LIN {X -0.030,Y -605.100,Z 1297.595,A 0.000,B 0.000,C 90.000,E1 143.050} C_DIS
LIN {X -0.184,Y -608.244,Z 1297.593,A 0.000,B 0.000,C 90.000,E1 142.683} C_DIS
LIN {X 0.115,Y -612.176,Z 1297.590,A 0.000,B 0.000,C 90.000,E1 142.145} C_DIS
LIN {X -0.312,Y -616.700,Z 1297.586,A 0.000,B 0.000,C 90.000,E1 141.537} C_DIS
LIN {X -0.216,Y -620.888,Z 1297.583,A 0.000,B 0.000,C 90.000,E1 140.884} C_DIS
LIN {X 0.278,Y -625.462,Z 1297.578,A 0.000,B 0.000,C 90.000,E1 140.070} C_DIS
LIN {X -0.003,Y -628.392,Z 1297.576,A 0.000,B 0.000,C 90.000,E1 139.585} C_DIS
LIN {X 0.188,Y -631.713,Z 1297.572,A 0.000,B 0.000,C 90.000,E1 138.933} C_DIS
LIN {X 0.321,Y -635.448,Z 1297.568,A 0.000,B 0.000,C 90.000,E1 138.162} C_DIS
LIN {X -0.415,Y -638.910,Z 1297.564,A 0.000,B 0.000,C 90.000,E1 137.472} C_DIS
LIN {X -0.130,Y -641.202,Z 1297.561,A 0.000,B 0.000,C 90.000,E1 136.944} C_DIS
LIN {X 0.323,Y -647.787,Z 1297.552,A 0.000,B 0.000,C 90.000,E1 135.405} C_DIS
LIN {X 0.041,Y -653.046,Z 1297.546,A 0.000,B 0.000,C 90.000,E1 134.190} C_DIS
LIN {X 0.316,Y -658.199,Z 1297.539,A 0.000,B 0.000,C 90.000,E1 132.933} C_DIS
LIN {X -0.258,Y -663.302,Z 1297.532,A 0.000,B 0.000,C 90.000,E1 131.757} C_DIS
LIN {X 0.194,Y -666.234,Z 1297.528,A 0.000,B 0.000,C 90.000,E1 130.987} C_DIS
LIN {X 0.237,Y -669.954,Z 1297.522,A 0.000,B 0.000,C 90.000,E1 130.011} C_DIS
LIN {X -0.092,Y -674.260,Z 1297.516,A 0.000,B 0.000,C 90.000,E1 128.830} C_DIS
LIN {X 0.179,Y -678.263,Z 1297.509,A 0.000,B 0.000,C 90.000,E1 127.604} C_DIS
LIN {X -0.045,Y -681.139,Z 1297.504,A 0.000,B 0.000,C 90.000,E1 126.664} C_DIS
LIN {X -0.238,Y -683.829,Z 1297.498,A 0.000,B 0.000,C 90.000,E1 125.724} C_DIS
LIN {X 0.153,Y -686.315,Z 1297.493,A 0.000,B 0.000,C 90.000,E1 124.739} C_DIS
LIN {X -0.013,Y -688.024,Z 1297.489,A 0.000,B 0.000,C 90.000,E1 124.040} C_DIS
LIN {X 0.045,Y -690.041,Z 1297.484,A 0.000,B 0.000,C 90.000,E1 123.086} C_DIS
LIN {X -0.092,Y -691.353,Z 1297.480,A 0.000,B 0.000,C 90.000,E1 122.388} C_DIS
LIN {X -0.359,Y -692.948,Z 1297.475,A 0.000,B 0.000,C 90.000,E1 121.465} C_DIS
LIN {X 0.244,Y -695.108,Z 1297.467,A 0.000,B 0.000,C 90.000,E1 120.001} C_DIS
LIN {X -0.217,Y -696.091,Z 1297.463,A 0.000,B 0.000,C 90.000,E1 119.333} C_DIS
LIN {X 0.194,Y -697.188,Z 1297.458,A 0.000,B 0.000,C 90.000,E1 118.359} C_DIS
LIN {X 0.359,Y -697.753,Z 1297.454,A 0.000,B 0.000,C 90.000,E1 117.641} C_DIS
LIN {X 0.210,Y -698.075,Z 1297.450,A 0.000,B 0.000,C 90.000,E1 116.950} C_DIS
LIN {X 0.018,Y -698.206,Z 1297.445,A 0.000,B 0.000,C 90.000,E1 116.027} C_DIS
LIN {X -0.122,Y -697.858,Z 1297.441,A 0.000,B 0.000,C 90.000,E1 115.335} C_DIS
LIN {X 0.107,Y -697.472,Z 1297.438,A 0.000,B 0.000,C 90.000,E1 114.847} C_DIS
LIN {X -0.004,Y -696.661,Z 1297.436,A 0.000,B 0.000,C 90.000,E1 114.387} C_DIS
LIN {X -0.032,Y -696.081,Z 1297.434,A 0.000,B 0.000,C 90.000,E1 114.155} C_DIS
LIN {X -0.157,Y -694.510,Z 1297.432,A 0.000,B 0.000,C 90.000,E1 113.695} C_DIS
LIN {X -0.033,Y -693.891,Z 1297.431,A 0.000,B 0.000,C 90.000,E1 113.567} C_DIS
LIN {X 0.179,Y -690.653,Z 1297.428,A 0.000,B 0.000,C 90.000,E1 113.078} C_DIS
LIN {X 0.298,Y -689.612,Z 1297.428,A 0.000,B 0.000,C 90.000,E1 112.950} C_DIS
LIN {X 0.145,Y -688.043,Z 1297.427,A 0.000,B 0.000,C 90.000,E1 112.845} C_DIS
LIN {X 0.031,Y -682.035,Z 1297.425,A 0.000,B 0.000,C 90.000,E1 112.461} C_DIS
LIN {X -0.099,Y -679.841,Z 1297.424,A 0.000,B 0.000,C 90.000,E1 112.386} C_DIS
LIN {X -0.135,Y -675.300,Z 1297.424,A 0.000,B 0.000,C 90.000,E1 112.259} C_DIS
LIN {X 0.009,Y -671.699,Z 1297.423,A 0.000,B 0.000,C 90.000,E1 112.153} C_DIS
LIN {X -0.191,Y -663.966,Z 1297.423,A 0.000,B 0.000,C 90.000,E1 112.078} C_DIS
LIN {X 0.309,Y -662.814,Z 1297.423,A 0.000,B 0.000,C 90.000,E1 112.025} C_DIS
LIN {X 0.251,Y -658.276,Z 1297.422,A 0.000,B 0.000,C 90.000,E1 112.025} C_DIS
LIN {X 0.138,Y -656.155,Z 1297.422,A 0.000,B 0.000,C 90.000,E1 112.025} C_DIS
LIN {X 0.082,Y -651.599,Z 1297.422,A 0.000,B 0.000,C 90.000,E1 112.025} C_DIS
LIN {X -0.029,Y -647.834,Z 1297.422,A 0.000,B 0.000,C 90.000,E1 112.025} C_DIS
LIN {X 0.046,Y -643.398,Z 1297.422,A 0.000,B 0.000,C 90.000,E1 111.972} C_DIS
LIN {X -0.186,Y -640.160,Z 1297.422,A 0.000,B 0.000,C 90.000,E1 111.897} C_DIS
LIN {X -0.223,Y -640.102,Z 1297.422,A 0.000,B 0.000,C 90.000,E1 111.897} C_DIS
LIN {X -0.025,Y -641.829,Z 1297.420,A 0.000,B 0.000,C 90.000,E1 111.535} C_DIS
LIN {X -0.231,Y -645.606,Z 1297.417,A 0.000,B 0.000,C 90.000,E1 111.046} C_DIS
LIN {X -0.292,Y -650.402,Z 1297.413,A 0.000,B 0.000,C 90.000,E1 110.429} C_DIS
LIN {X 0.343,Y -655.261,Z 1297.409,A 0.000,B 0.000,C 90.000,E1 109.631} C_DIS
LIN {X 0.142,Y -658.719,Z 1297.406,A 0.000,B 0.000,C 90.000,E1 109.033} C_DIS
LIN {X 0.079,Y -660.661,Z 1297.404,A 0.000,B 0.000,C 90.000,E1 108.671} C_DIS
LIN {X -0.024,Y -664.077,Z 1297.400,A 0.000,B 0.000,C 90.000,E1 107.946} C_DIS
LIN {X -0.098,Y -667.037,Z 1297.396,A 0.000,B 0.000,C 90.000,E1 107.221} C_DIS
LIN {X -0.069,Y -668.785,Z 1297.393,A 0.000,B 0.000,C 90.000,E1 106.732} C_DIS
LIN {X -0.294,Y -671.049,Z 1297.389,A 0.000,B 0.000,C 90.000,E1 106.024} C_DIS
LIN {X 0.336,Y -672.875,Z 1297.385,A 0.000,B 0.000,C 90.000,E1 105.245} C_DIS
LIN {X 0.215,Y -673.985,Z 1297.382,A 0.000,B 0.000,C 90.000,E1 104.773} C_DIS
LIN {X 0.048,Y -675.282,Z 1297.378,A 0.000,B 0.000,C 90.000,E1 104.064} C_DIS
LIN {X -0.057,Y -676.027,Z 1297.375,A 0.000,B 0.000,C 90.000,E1 103.592} C_DIS
LIN {X -0.206,Y -676.735,Z 1297.372,A 0.000,B 0.000,C 90.000,E1 102.883} C_DIS
LIN {X 0.308,Y -677.148,Z 1297.368,A 0.000,B 0.000,C 90.000,E1 102.119} C_DIS
LIN {X 0.026,Y -677.120,Z 1297.364,A 0.000,B 0.000,C 90.000,E1 101.422} C_DIS
LIN {X -0.072,Y -676.885,Z 1297.361,A 0.000,B 0.000,C 90.000,E1 100.950} C_DIS
LIN {X 0.313,Y -676.130,Z 1297.357,A 0.000,B 0.000,C 90.000,E1 100.197} C_DIS
LIN {X 0.202,Y -675.321,Z 1297.354,A 0.000,B 0.000,C 90.000,E1 99.726} C_DIS
LIN {X -0.029,Y -674.316,Z 1297.352,A 0.000,B 0.000,C 90.000,E1 99.265} C_DIS
LIN {X -0.263,Y -672.938,Z 1297.349,A 0.000,B 0.000,C 90.000,E1 98.803} C_DIS
LIN {X 0.260,Y -671.215,Z 1297.346,A 0.000,B 0.000,C 90.000,E1 98.276} C_DIS
LIN {X 0.008,Y -669.140,Z 1297.344,A 0.000,B 0.000,C 90.000,E1 97.814} C_DIS
LIN {X 0.230,Y -665.625,Z 1297.339,A 0.000,B 0.000,C 90.000,E1 97.068} C_DIS
LIN {X -0.071,Y -662.116,Z 1297.336,A 0.000,B 0.000,C 90.000,E1 96.486} C_DIS
LIN {X 0.276,Y -659.164,Z 1297.333,A 0.000,B 0.000,C 90.000,E1 95.967} C_DIS
LIN {X -0.085,Y -655.897,Z 1297.331,A 0.000,B 0.000,C 90.000,E1 95.511} C_DIS
LIN {X 0.147,Y -651.287,Z 1297.327,A 0.000,B 0.000,C 90.000,E1 94.878} C_DIS
LIN {X -0.215,Y -647.287,Z 1297.324,A 0.000,B 0.000,C 90.000,E1 94.416} C_DIS
LIN {X 0.310,Y -639.394,Z 1297.320,A 0.000,B 0.000,C 90.000,E1 93.498} C_DIS
LIN {X 0.036,Y -629.758,Z 1297.314,A 0.000,B 0.000,C 90.000,E1 92.522} C_DIS
LIN {X -0.068,Y -626.245,Z 1297.312,A 0.000,B 0.000,C 90.000,E1 92.178} C_DIS
LIN {X 0.266,Y -621.098,Z 1297.309,A 0.000,B 0.000,C 90.000,E1 91.661} C_DIS
LIN {X 0.159,Y -615.486,Z 1297.307,A 0.000,B 0.000,C 90.000,E1 91.203} C_DIS
LIN {X 0.033,Y -608.005,Z 1297.304,A 0.000,B 0.000,C 90.000,E1 90.688} C_DIS
LIN {X 0.125,Y -601.709,Z 1297.302,A 0.000,B 0.000,C 90.000,E1 90.286} C_DIS
LIN {X -0.026,Y -595.069,Z 1297.300,A 0.000,B 0.000,C 90.000,E1 89.943} C_DIS
LIN {X 0.231,Y -588.114,Z 1297.298,A 0.000,B 0.000,C 90.000,E1 89.599} C_DIS
LIN {X -0.248,Y -578.956,Z 1297.296,A 0.000,B 0.000,C 90.000,E1 89.312} C_DIS
LIN {X 0.252,Y -575.828,Z 1297.295,A 0.000,B 0.000,C 90.000,E1 89.141} C_DIS
LIN {X 0.201,Y -571.918,Z 1297.294,A 0.000,B 0.000,C 90.000,E1 88.969} C_DIS
LIN {X 0.184,Y -570.507,Z 1297.294,A 0.000,B 0.000,C 90.000,E1 88.854} C_DIS
LIN {X 0.147,Y -570.464,Z 1297.294,A 0.000,B 0.000,C 90.000,E1 88.854} C_DIS
LIN {X -0.051,Y -569.912,Z 1297.293,A 0.000,B 0.000,C 90.000,E1 88.740} C_DIS
LIN {X -0.187,Y -569.791,Z 1297.291,A 0.000,B 0.000,C 90.000,E1 88.339} C_DIS
LIN {X 0.170,Y -572.199,Z 1297.274,A 0.000,B 0.000,C 90.000,E1 85.298} C_DIS
LIN {X 0.146,Y -574.318,Z 1297.263,A 0.000,B 0.000,C 90.000,E1 83.394} C_DIS
LIN {X 0.180,Y -576.536,Z 1297.253,A 0.000,B 0.000,C 90.000,E1 81.489} C_DIS
LIN {X 0.225,Y -578.520,Z 1297.244,A 0.000,B 0.000,C 90.000,E1 79.859} C_DIS
LIN {X -0.137,Y -579.666,Z 1297.238,A 0.000,B 0.000,C 90.000,E1 78.814} C_DIS
LIN {X -0.146,Y -580.931,Z 1297.230,A 0.000,B 0.000,C 90.000,E1 77.465} C_DIS
LIN {X -0.136,Y -582.120,Z 1297.223,A 0.000,B 0.000,C 90.000,E1 76.117} C_DIS
LIN {X -0.305,Y -583.309,Z 1297.214,A 0.000,B 0.000,C 90.000,E1 74.519} C_DIS
LIN {X 0.039,Y -584.186,Z 1297.206,A 0.000,B 0.000,C 90.000,E1 73.142} C_DIS
LIN {X 0.066,Y -585.263,Z 1297.198,A 0.000,B 0.000,C 90.000,E1 71.529} C_DIS
LIN {X -0.145,Y -585.939,Z 1297.192,A 0.000,B 0.000,C 90.000,E1 70.477} C_DIS
LIN {X 0.093,Y -586.922,Z 1297.183,A 0.000,B 0.000,C 90.000,E1 68.847} C_DIS
LIN {X -0.246,Y -588.232,Z 1297.171,A 0.000,B 0.000,C 90.000,E1 66.741} C_DIS
LIN {X 0.150,Y -589.357,Z 1297.162,A 0.000,B 0.000,C 90.000,E1 65.101} C_DIS
LIN {X 0.041,Y -590.511,Z 1297.153,A 0.000,B 0.000,C 90.000,E1 63.512} C_DIS
LIN {X 0.120,Y -592.082,Z 1297.143,A 0.000,B 0.000,C 90.000,E1 61.641} C_DIS
LIN {X -0.095,Y -593.382,Z 1297.135,A 0.000,B 0.000,C 90.000,E1 60.333} C_DIS
LIN {X 0.009,Y -594.730,Z 1297.128,A 0.000,B 0.000,C 90.000,E1 58.997} C_DIS
LIN {X 0.035,Y -596.340,Z 1297.119,A 0.000,B 0.000,C 90.000,E1 57.406} C_DIS
LIN {X 0.107,Y -597.490,Z 1297.113,A 0.000,B 0.000,C 90.000,E1 56.342} C_DIS
LIN {X 0.109,Y -598.850,Z 1297.106,A 0.000,B 0.000,C 90.000,E1 55.022} C_DIS
LIN {X -0.111,Y -600.333,Z 1297.097,A 0.000,B 0.000,C 90.000,E1 53.463} C_DIS
LIN {X -0.311,Y -601.668,Z 1297.088,A 0.000,B 0.000,C 90.000,E1 51.904} C_DIS
LIN {X 0.217,Y -602.537,Z 1297.082,A 0.000,B 0.000,C 90.000,E1 50.803} C_DIS
LIN {X -0.057,Y -603.473,Z 1297.074,A 0.000,B 0.000,C 90.000,E1 49.256} C_DIS
LIN {X -0.016,Y -603.749,Z 1297.071,A 0.000,B 0.000,C 90.000,E1 48.728} C_DIS
LIN {X 0.226,Y -603.990,Z 1297.066,A 0.000,B 0.000,C 90.000,E1 47.919} C_DIS
LIN {X -0.084,Y -604.366,Z 1297.058,A 0.000,B 0.000,C 90.000,E1 46.377} C_DIS
LIN {X -0.017,Y -604.520,Z 1297.052,A 0.000,B 0.000,C 90.000,E1 45.324} C_DIS
LIN {X 0.055,Y -604.463,Z 1297.046,A 0.000,B 0.000,C 90.000,E1 44.271} C_DIS
LIN {X -0.080,Y -604.111,Z 1297.039,A 0.000,B 0.000,C 90.000,E1 42.975} C_DIS
LIN {X 0.008,Y -603.839,Z 1297.033,A 0.000,B 0.000,C 90.000,E1 41.919} C_DIS
LIN {X -0.149,Y -603.531,Z 1297.029,A 0.000,B 0.000,C 90.000,E1 41.148} C_DIS
LIN {X 0.233,Y -602.687,Z 1297.018,A 0.000,B 0.000,C 90.000,E1 39.277} C_DIS
LIN {X -0.071,Y -602.062,Z 1297.013,A 0.000,B 0.000,C 90.000,E1 38.257} C_DIS
LIN {X -0.134,Y -600.871,Z 1297.005,A 0.000,B 0.000,C 90.000,E1 36.950} C_DIS
LIN {X 0.016,Y -599.578,Z 1296.999,A 0.000,B 0.000,C 90.000,E1 35.884} C_DIS
LIN {X 0.145,Y -598.081,Z 1296.994,A 0.000,B 0.000,C 90.000,E1 34.818} C_DIS
LIN {X 0.135,Y -595.738,Z 1296.986,A 0.000,B 0.000,C 90.000,E1 33.499} C_DIS
LIN {X -0.349,Y -594.062,Z 1296.982,A 0.000,B 0.000,C 90.000,E1 32.752} C_DIS
LIN {X -0.240,Y -592.810,Z 1296.979,A 0.000,B 0.000,C 90.000,E1 32.212} C_DIS
LIN {X 0.061,Y -590.612,Z 1296.974,A 0.000,B 0.000,C 90.000,E1 31.386} C_DIS
LIN {X 0.029,Y -588.195,Z 1296.970,A 0.000,B 0.000,C 90.000,E1 30.590} C_DIS
LIN {X -0.028,Y -585.262,Z 1296.966,A 0.000,B 0.000,C 90.000,E1 29.795} C_DIS
LIN {X -0.272,Y -583.140,Z 1296.963,A 0.000,B 0.000,C 90.000,E1 29.283} C_DIS
LIN {X 0.131,Y -579.545,Z 1296.958,A 0.000,B 0.000,C 90.000,E1 28.437} C_DIS
LIN {X 0.197,Y -577.635,Z 1296.956,A 0.000,B 0.000,C 90.000,E1 28.025} C_DIS
LIN {X -0.171,Y -574.033,Z 1296.952,A 0.000,B 0.000,C 90.000,E1 27.385} C_DIS
LIN {X 0.117,Y -569.415,Z 1296.948,A 0.000,B 0.000,C 90.000,E1 26.539} C_DIS
LIN {X 0.100,Y -564.275,Z 1296.943,A 0.000,B 0.000,C 90.000,E1 25.720} C_DIS
LIN {X 0.228,Y -560.522,Z 1296.940,A 0.000,B 0.000,C 90.000,E1 25.155} C_DIS
LIN {X -0.165,Y -556.580,Z 1296.937,A 0.000,B 0.000,C 90.000,E1 24.643} C_DIS
LIN {X -0.089,Y -552.362,Z 1296.934,A 0.000,B 0.000,C 90.000,E1 24.079} C_DIS
LIN {X 0.074,Y -549.001,Z 1296.931,A 0.000,B 0.000,C 90.000,E1 23.643} C_DIS
LIN {X 0.095,Y -544.241,Z 1296.928,A 0.000,B 0.000,C 90.000,E1 23.078} C_DIS
LIN {X -0.107,Y -537.173,Z 1296.924,A 0.000,B 0.000,C 90.000,E1 22.280} C_DIS
LIN {X 0.213,Y -530.692,Z 1296.920,A 0.000,B 0.000,C 90.000,E1 21.535} C_DIS
LIN {X -0.227,Y -521.569,Z 1296.914,A 0.000,B 0.000,C 90.000,E1 20.610} C_DIS
LIN {X 0.161,Y -512.498,Z 1296.909,A 0.000,B 0.000,C 90.000,E1 19.631} C_DIS
LIN {X 0.116,Y -504.674,Z 1296.905,A 0.000,B 0.000,C 90.000,E1 18.852} C_DIS
LIN {X -0.143,Y -495.008,Z 1296.900,A 0.000,B 0.000,C 90.000,E1 17.928} C_DIS
LIN {X -0.016,Y -483.925,Z 1296.894,A 0.000,B 0.000,C 90.000,E1 16.858} C_DIS
LIN {X -0.090,Y -473.781,Z 1296.889,A 0.000,B 0.000,C 90.000,E1 15.953} C_DIS
LIN {X 0.015,Y -463.432,Z 1296.883,A 0.000,B 0.000,C 90.000,E1 15.009} C_DIS
LIN {X -0.079,Y -447.415,Z 1296.875,A 0.000,B 0.000,C 90.000,E1 13.536} C_DIS
LIN {X -0.029,Y -427.454,Z 1296.864,A 0.000,B 0.000,C 90.000,E1 11.535} C_DIS
LIN {X -0.194,Y -408.819,Z 1296.853,A 0.000,B 0.000,C 90.000,E1 9.557} C_DIS
LIN {X 0.118,Y -400.386,Z 1296.848,A 0.000,B 0.000,C 90.000,E1 8.568} C_DIS
LIN {X -0.145,Y -396.849,Z 1296.845,A 0.000,B 0.000,C 90.000,E1 8.163} C_DIS
LIN {X 0.146,Y -395.306,Z 1296.844,A 0.000,B 0.000,C 90.000,E1 7.814} C_DIS
LIN {X 0.108,Y -395.286,Z 1296.844,A 0.000,B 0.000,C 90.000,E1 7.814} C_DIS
LIN {X 0.106,Y -396.353,Z 1296.843,A 0.000,B 0.000,C 90.000,E1 7.644} C_DIS
LIN {X 0.203,Y -398.732,Z 1296.841,A 0.000,B 0.000,C 90.000,E1 7.409} C_DIS
LIN {X 0.001,Y -400.479,Z 1296.841,A 0.000,B 0.000,C 90.000,E1 7.296} C_DIS
LIN {X -0.011,Y -406.290,Z 1296.839,A 0.000,B 0.000,C 90.000,E1 6.947} C_DIS
LIN {X -0.066,Y -412.341,Z 1296.837,A 0.000,B 0.000,C 90.000,E1 6.606} C_DIS
LIN {X -0.215,Y -418.697,Z 1296.834,A 0.000,B 0.000,C 90.000,E1 6.201} C_DIS
LIN {X -0.169,Y -423.565,Z 1296.832,A 0.000,B 0.000,C 90.000,E1 5.853} C_DIS
LIN {X 0.116,Y -432.755,Z 1296.828,A 0.000,B 0.000,C 90.000,E1 5.106} C_DIS
LIN {X -0.081,Y -437.351,Z 1296.826,A 0.000,B 0.000,C 90.000,E1 4.759} C_DIS
LIN {X 0.069,Y -446.607,Z 1296.822,A 0.000,B 0.000,C 90.000,E1 3.955} C_DIS
LIN {X -0.154,Y -453.959,Z 1296.818,A 0.000,B 0.000,C 90.000,E1 3.326} C_DIS
LIN {X -0.200,Y -461.137,Z 1296.815,A 0.000,B 0.000,C 90.000,E1 2.636} C_DIS
LIN {X -0.203,Y -466.756,Z 1296.811,A 0.000,B 0.000,C 90.000,E1 2.064} C_DIS
LIN {X -0.154,Y -473.457,Z 1296.807,A 0.000,B 0.000,C 90.000,E1 1.318} C_DIS
LIN {X -0.036,Y -478.418,Z 1296.804,A 0.000,B 0.000,C 90.000,E1 0.688} C_DIS
LIN {X -0.098,Y -482.096,Z 1296.801,A 0.000,B 0.000,C 90.000,E1 0.229} C_DIS
LIN {X 0.004,Y -487.458,Z 1296.797,A 0.000,B 0.000,C 90.000,E1 359.484} C_DIS
LIN {X 0.000,Y -493.503,Z 1296.792,A 0.000,B 0.000,C 90.000,E1 358.568} C_DIS
LIN {X 0.216,Y -497.387,Z 1296.789,A 0.000,B 0.000,C 90.000,E1 357.936} C_DIS
LIN {X -0.179,Y -502.545,Z 1296.784,A 0.000,B 0.000,C 90.000,E1 357.078} C_DIS
LIN {X -0.193,Y -506.613,Z 1296.780,A 0.000,B 0.000,C 90.000,E1 356.331} C_DIS
LIN {X -0.169,Y -510.442,Z 1296.775,A 0.000,B 0.000,C 90.000,E1 355.584} C_DIS
LIN {X -0.107,Y -514.022,Z 1296.771,A 0.000,B 0.000,C 90.000,E1 354.837} C_DIS
LIN {X -0.230,Y -516.705,Z 1296.768,A 0.000,B 0.000,C 90.000,E1 354.261} C_DIS
LIN {X -0.116,Y -519.816,Z 1296.764,A 0.000,B 0.000,C 90.000,E1 353.514} C_DIS
LIN {X -0.209,Y -523.311,Z 1296.759,A 0.000,B 0.000,C 90.000,E1 352.648} C_DIS
LIN {X -0.265,Y -526.526,Z 1296.754,A 0.000,B 0.000,C 90.000,E1 351.781} C_DIS
LIN {X -0.264,Y -530.268,Z 1296.748,A 0.000,B 0.000,C 90.000,E1 350.622} C_DIS
LIN {X -0.158,Y -532.820,Z 1296.743,A 0.000,B 0.000,C 90.000,E1 349.746} C_DIS
LIN {X 0.033,Y -535.871,Z 1296.737,A 0.000,B 0.000,C 90.000,E1 348.578} C_DIS
LIN {X 0.207,Y -537.895,Z 1296.732,A 0.000,B 0.000,C 90.000,E1 347.701} C_DIS
LIN {X -0.125,Y -539.628,Z 1296.727,A 0.000,B 0.000,C 90.000,E1 346.881} C_DIS
LIN {X -0.240,Y -541.622,Z 1296.721,A 0.000,B 0.000,C 90.000,E1 345.755} C_DIS
LIN {X -0.093,Y -542.514,Z 1296.718,A 0.000,B 0.000,C 90.000,E1 345.172} C_DIS
LIN {X -0.249,Y -543.546,Z 1296.713,A 0.000,B 0.000,C 90.000,E1 344.338} C_DIS
LIN {X 0.129,Y -544.404,Z 1296.708,A 0.000,B 0.000,C 90.000,E1 343.449} C_DIS
LIN {X 0.154,Y -545.096,Z 1296.703,A 0.000,B 0.000,C 90.000,E1 342.598} C_DIS
LIN {X 0.024,Y -545.466,Z 1296.699,A 0.000,B 0.000,C 90.000,E1 341.764} C_DIS
LIN {X 0.068,Y -545.510,Z 1296.694,A 0.000,B 0.000,C 90.000,E1 340.913} C_DIS
LIN {X 0.114,Y -545.290,Z 1296.689,A 0.000,B 0.000,C 90.000,E1 340.061} C_DIS
LIN {X -0.091,Y -544.955,Z 1296.686,A 0.000,B 0.000,C 90.000,E1 339.518} C_DIS
LIN {X 0.142,Y -544.243,Z 1296.682,A 0.000,B 0.000,C 90.000,E1 338.646} C_DIS
LIN {X -0.318,Y -543.959,Z 1296.680,A 0.000,B 0.000,C 90.000,E1 338.411} C_DIS
LIN {X 0.122,Y -541.386,Z 1296.671,A 0.000,B 0.000,C 90.000,E1 336.666} C_DIS
LIN {X -0.172,Y -539.466,Z 1296.666,A 0.000,B 0.000,C 90.000,E1 335.845} C_DIS
LIN {X 0.276,Y -537.998,Z 1296.663,A 0.000,B 0.000,C 90.000,E1 335.229} C_DIS
LIN {X -0.055,Y -535.645,Z 1296.658,A 0.000,B 0.000,C 90.000,E1 334.409} C_DIS
LIN {X 0.018,Y -531.934,Z 1296.651,A 0.000,B 0.000,C 90.000,E1 333.256} C_DIS
LIN {X 0.037,Y -528.228,Z 1296.645,A 0.000,B 0.000,C 90.000,E1 332.103} C_DIS
LIN {X -0.158,Y -525.084,Z 1296.640,A 0.000,B 0.000,C 90.000,E1 331.257} C_DIS
LIN {X 0.030,Y -522.114,Z 1296.636,A 0.000,B 0.000,C 90.000,E1 330.511} C_DIS
LIN {X -0.067,Y -518.892,Z 1296.632,A 0.000,B 0.000,C 90.000,E1 329.793} C_DIS
LIN {X 0.162,Y -513.915,Z 1296.626,A 0.000,B 0.000,C 90.000,E1 328.742} C_DIS
LIN {X 0.247,Y -510.206,Z 1296.622,A 0.000,B 0.000,C 90.000,E1 327.995} C_DIS
LIN {X 0.004,Y -504.500,Z 1296.616,A 0.000,B 0.000,C 90.000,E1 326.834} C_DIS
LIN {X 0.086,Y -500.941,Z 1296.611,A 0.000,B 0.000,C 90.000,E1 325.928} C_DIS
LIN {X -0.031,Y -499.901,Z 1296.609,A 0.000,B 0.000,C 90.000,E1 325.642} C_DIS
LIN {X -0.277,Y -497.630,Z 1296.604,A 0.000,B 0.000,C 90.000,E1 324.769} C_DIS
LIN {X 0.023,Y -496.098,Z 1296.599,A 0.000,B 0.000,C 90.000,E1 323.829} C_DIS
LIN {X 0.034,Y -494.696,Z 1296.591,A 0.000,B 0.000,C 90.000,E1 322.316} C_DIS
LIN {X 0.162,Y -494.242,Z 1296.584,A 0.000,B 0.000,C 90.000,E1 321.090} C_DIS
LIN {X -0.205,Y -494.321,Z 1296.569,A 0.000,B 0.000,C 90.000,E1 318.405} C_DIS
LIN {X 0.021,Y -494.491,Z 1296.560,A 0.000,B 0.000,C 90.000,E1 316.863} C_DIS
LIN {X 0.048,Y -494.625,Z 1296.554,A 0.000,B 0.000,C 90.000,E1 315.648} C_DIS
LIN {X -0.101,Y -494.374,Z 1296.549,A 0.000,B 0.000,C 90.000,E1 314.757} C_DIS
LIN {X 0.263,Y -493.971,Z 1296.545,A 0.000,B 0.000,C 90.000,E1 314.109} C_DIS
LIN {X -0.075,Y -493.312,Z 1296.542,A 0.000,B 0.000,C 90.000,E1 313.542} C_DIS
LIN {X 0.102,Y -492.831,Z 1296.540,A 0.000,B 0.000,C 90.000,E1 313.218} C_DIS
LIN {X -0.059,Y -492.218,Z 1296.539,A 0.000,B 0.000,C 90.000,E1 312.933} C_DIS
LIN {X 0.115,Y -491.395,Z 1296.537,A 0.000,B 0.000,C 90.000,E1 312.609} C_DIS
LIN {X 0.200,Y -490.846,Z 1296.536,A 0.000,B 0.000,C 90.000,E1 312.447} C_DIS
LIN {X -0.046,Y -490.118,Z 1296.535,A 0.000,B 0.000,C 90.000,E1 312.324} C_DIS
LIN {X 0.229,Y -480.831,Z 1296.528,A 0.000,B 0.000,C 90.000,E1 311.067} C_DIS
LIN {X 0.080,Y -463.374,Z 1296.515,A 0.000,B 0.000,C 90.000,E1 308.588} C_DIS
LIN {X 0.214,Y -447.591,Z 1296.500,A 0.000,B 0.000,C 90.000,E1 306.011} C_DIS
LIN {X 0.052,Y -432.542,Z 1296.485,A 0.000,B 0.000,C 90.000,E1 303.245} C_DIS
LIN {X -0.081,Y -419.160,Z 1296.469,A 0.000,B 0.000,C 90.000,E1 300.413} C_DIS
LIN {X -0.139,Y -407.347,Z 1296.453,A 0.000,B 0.000,C 90.000,E1 297.513} C_DIS
LIN {X -0.160,Y -399.156,Z 1296.440,A 0.000,B 0.000,C 90.000,E1 295.207} C_DIS
LIN {X 0.163,Y -399.138,Z 1296.440,A 0.000,B 0.000,C 90.000,E1 295.155} C_DIS
LIN {X 0.076,Y -401.525,Z 1296.427,A 0.000,B 0.000,C 90.000,E1 292.770} C_DIS
LIN {X 0.109,Y -401.877,Z 1296.421,A 0.000,B 0.000,C 90.000,E1 291.716} C_DIS
LIN {X -0.168,Y -404.596,Z 1296.396,A 0.000,B 0.000,C 90.000,E1 287.221} C_DIS
LIN {X -0.068,Y -404.758,Z 1296.394,A 0.000,B 0.000,C 90.000,E1 286.858} C_DIS
LIN {X -0.161,Y -406.059,Z 1296.365,A 0.000,B 0.000,C 90.000,E1 281.658} C_DIS
LIN {X -0.071,Y -406.123,Z 1296.363,A 0.000,B 0.000,C 90.000,E1 281.299} C_DIS
LIN {X -0.041,Y -405.663,Z 1296.334,A 0.000,B 0.000,C 90.000,E1 276.087} C_DIS
LIN {X -0.036,Y -405.577,Z 1296.332,A 0.000,B 0.000,C 90.000,E1 275.739} C_DIS
LIN {X 0.038,Y -403.537,Z 1296.305,A 0.000,B 0.000,C 90.000,E1 270.859} C_DIS
LIN {X -0.027,Y -403.004,Z 1296.301,A 0.000,B 0.000,C 90.000,E1 270.172} C_DIS
LIN {X 0.193,Y -398.991,Z 1296.272,A 0.000,B 0.000,C 90.000,E1 264.894} C_DIS
LIN {X -0.043,Y -392.898,Z 1296.240,A 0.000,B 0.000,C 90.000,E1 259.285} C_DIS
LIN {X -0.096,Y -391.246,Z 1296.235,A 0.000,B 0.000,C 90.000,E1 258.229} C_DIS
LIN {X 0.098,Y -385.339,Z 1296.209,A 0.000,B 0.000,C 90.000,E1 253.559} C_DIS
LIN {X 0.120,Y -384.904,Z 1296.207,A 0.000,B 0.000,C 90.000,E1 253.196} C_DIS
LIN {X 0.120,Y -381.655,Z 1296.196,A 0.000,B 0.000,C 90.000,E1 251.329} C_DIS
LIN {X 0.082,Y -381.665,Z 1296.196,A 0.000,B 0.000,C 90.000,E1 251.329} C_DIS
LIN {X 0.178,Y -390.790,Z 1296.177,A 0.000,B 0.000,C 90.000,E1 247.794} C_DIS
LIN {X -0.208,Y -400.781,Z 1296.159,A 0.000,B 0.000,C 90.000,E1 244.665} C_DIS
LIN {X -0.081,Y -411.695,Z 1296.143,A 0.000,B 0.000,C 90.000,E1 241.691} C_DIS
LIN {X -0.078,Y -424.135,Z 1296.127,A 0.000,B 0.000,C 90.000,E1 238.791} C_DIS
LIN {X 0.086,Y -438.192,Z 1296.111,A 0.000,B 0.000,C 90.000,E1 235.928} C_DIS
LIN {X -0.078,Y -452.017,Z 1296.097,A 0.000,B 0.000,C 90.000,E1 233.497} C_DIS
LIN {X -0.087,Y -452.738,Z 1296.096,A 0.000,B 0.000,C 90.000,E1 233.336} C_DIS
LIN {X 0.267,Y -453.254,Z 1296.095,A 0.000,B 0.000,C 90.000,E1 233.130} C_DIS
LIN {X -0.016,Y -453.988,Z 1296.094,A 0.000,B 0.000,C 90.000,E1 232.844} C_DIS
LIN {X -0.298,Y -454.503,Z 1296.092,A 0.000,B 0.000,C 90.000,E1 232.557} C_DIS
LIN {X -0.217,Y -455.156,Z 1296.088,A 0.000,B 0.000,C 90.000,E1 231.904} C_DIS
LIN {X -0.120,Y -455.578,Z 1296.083,A 0.000,B 0.000,C 90.000,E1 230.928} C_DIS
LIN {X -0.011,Y -455.552,Z 1296.078,A 0.000,B 0.000,C 90.000,E1 229.952} C_DIS
LIN {X -0.086,Y -454.876,Z 1296.065,A 0.000,B 0.000,C 90.000,E1 227.715} C_DIS
LIN {X -0.270,Y -454.436,Z 1296.054,A 0.000,B 0.000,C 90.000,E1 225.810} C_DIS
LIN {X -0.121,Y -454.299,Z 1296.042,A 0.000,B 0.000,C 90.000,E1 223.542} C_DIS
LIN {X 0.023,Y -455.854,Z 1296.013,A 0.000,B 0.000,C 90.000,E1 218.382} C_DIS
LIN {X 0.037,Y -457.124,Z 1296.003,A 0.000,B 0.000,C 90.000,E1 216.457} C_DIS
LIN {X -0.224,Y -459.810,Z 1295.985,A 0.000,B 0.000,C 90.000,E1 213.293} C_DIS
LIN {X 0.027,Y -463.273,Z 1295.967,A 0.000,B 0.000,C 90.000,E1 210.079} C_DIS
LIN {X 0.086,Y -465.311,Z 1295.958,A 0.000,B 0.000,C 90.000,E1 208.487} C_DIS
LIN {X -0.089,Y -469.122,Z 1295.943,A 0.000,B 0.000,C 90.000,E1 205.668} C_DIS
LIN {X 0.060,Y -471.422,Z 1295.934,A 0.000,B 0.000,C 90.000,E1 204.079} C_DIS
LIN {X 0.021,Y -474.125,Z 1295.923,A 0.000,B 0.000,C 90.000,E1 202.206} C_DIS
LIN {X -0.143,Y -476.966,Z 1295.913,A 0.000,B 0.000,C 90.000,E1 200.355} C_DIS
LIN {X 0.049,Y -479.406,Z 1295.904,A 0.000,B 0.000,C 90.000,E1 198.779} C_DIS
LIN {X 0.145,Y -481.900,Z 1295.896,A 0.000,B 0.000,C 90.000,E1 197.221} C_DIS
LIN {X -0.176,Y -484.438,Z 1295.887,A 0.000,B 0.000,C 90.000,E1 195.717} C_DIS
LIN {X -0.125,Y -486.910,Z 1295.879,A 0.000,B 0.000,C 90.000,E1 194.175} C_DIS
LIN {X -0.142,Y -489.429,Z 1295.870,A 0.000,B 0.000,C 90.000,E1 192.647} C_DIS
LIN {X 0.167,Y -492.369,Z 1295.860,A 0.000,B 0.000,C 90.000,E1 190.782} C_DIS
LIN {X 0.157,Y -494.834,Z 1295.852,A 0.000,B 0.000,C 90.000,E1 189.265} C_DIS
LIN {X 0.107,Y -497.287,Z 1295.843,A 0.000,B 0.000,C 90.000,E1 187.757} C_DIS
LIN {X -0.053,Y -500.128,Z 1295.833,A 0.000,B 0.000,C 90.000,E1 185.967} C_DIS
LIN {X 0.004,Y -501.996,Z 1295.827,A 0.000,B 0.000,C 90.000,E1 184.759} C_DIS
LIN {X 0.242,Y -505.046,Z 1295.815,A 0.000,B 0.000,C 90.000,E1 182.636} C_DIS
LIN {X -0.169,Y -506.619,Z 1295.808,A 0.000,B 0.000,C 90.000,E1 181.489} C_DIS
LIN {X -0.159,Y -508.417,Z 1295.800,A 0.000,B 0.000,C 90.000,E1 180.000} C_DIS
LIN {X -0.024,Y -509.682,Z 1295.793,A 0.000,B 0.000,C 90.000,E1 178.797} C_DIS
LIN {X 0.142,Y -510.735,Z 1295.787,A 0.000,B 0.000,C 90.000,E1 177.593} C_DIS
LIN {X -0.184,Y -511.719,Z 1295.780,A 0.000,B 0.000,C 90.000,E1 176.445} C_DIS
LIN {X 0.097,Y -512.241,Z 1295.775,A 0.000,B 0.000,C 90.000,E1 175.527} C_DIS
LIN {X -0.171,Y -512.768,Z 1295.769,A 0.000,B 0.000,C 90.000,E1 174.375} C_DIS
LIN {X 0.077,Y -512.987,Z 1295.762,A 0.000,B 0.000,C 90.000,E1 173.166} C_DIS
LIN {X -0.119,Y -512.937,Z 1295.756,A 0.000,B 0.000,C 90.000,E1 172.008} C_DIS
LIN {X 0.223,Y -512.634,Z 1295.751,A 0.000,B 0.000,C 90.000,E1 171.084} C_DIS
LIN {X 0.017,Y -511.872,Z 1295.744,A 0.000,B 0.000,C 90.000,E1 169.926} C_DIS
LIN {X -0.111,Y -510.857,Z 1295.738,A 0.000,B 0.000,C 90.000,E1 168.757} C_DIS
LIN {X -0.216,Y -509.724,Z 1295.733,A 0.000,B 0.000,C 90.000,E1 167.881} C_DIS
LIN {X -0.182,Y -508.876,Z 1295.729,A 0.000,B 0.000,C 90.000,E1 167.285} C_DIS
LIN {X 0.136,Y -506.863,Z 1295.723,A 0.000,B 0.000,C 90.000,E1 166.061} C_DIS
LIN {X 0.156,Y -505.632,Z 1295.719,A 0.000,B 0.000,C 90.000,E1 165.463} C_DIS
LIN {X 0.045,Y -503.186,Z 1295.713,A 0.000,B 0.000,C 90.000,E1 164.283} C_DIS
LIN {X 0.031,Y -500.598,Z 1295.706,A 0.000,B 0.000,C 90.000,E1 163.087} C_DIS
LIN {X 0.132,Y -497.598,Z 1295.699,A 0.000,B 0.000,C 90.000,E1 161.873} C_DIS
LIN {X 0.080,Y -493.755,Z 1295.691,A 0.000,B 0.000,C 90.000,E1 160.369} C_DIS
LIN {X 0.110,Y -489.657,Z 1295.683,A 0.000,B 0.000,C 90.000,E1 158.847} C_DIS
LIN {X -0.256,Y -487.784,Z 1295.677,A 0.000,B 0.000,C 90.000,E1 157.975} C_DIS
LIN {X -0.209,Y -487.143,Z 1295.674,A 0.000,B 0.000,C 90.000,E1 157.358} C_DIS
LIN {X -0.188,Y -487.149,Z 1295.672,A 0.000,B 0.000,C 90.000,E1 157.050} C_DIS
LIN {X -0.170,Y -487.657,Z 1295.671,A 0.000,B 0.000,C 90.000,E1 156.741} C_DIS
LIN {X -0.146,Y -489.766,Z 1295.667,A 0.000,B 0.000,C 90.000,E1 155.973} C_DIS
LIN {X 0.031,Y -491.600,Z 1295.665,A 0.000,B 0.000,C 90.000,E1 155.613} C_DIS
LIN {X -0.178,Y -493.182,Z 1295.664,A 0.000,B 0.000,C 90.000,E1 155.485} C_DIS
LIN {X 0.061,Y -494.422,Z 1295.663,A 0.000,B 0.000,C 90.000,E1 155.305} C_DIS
LIN {X 0.064,Y -495.469,Z 1295.662,A 0.000,B 0.000,C 90.000,E1 155.153} C_DIS
LIN {X -0.141,Y -496.751,Z 1295.661,A 0.000,B 0.000,C 90.000,E1 155.025} C_DIS
LIN {X 0.005,Y -498.389,Z 1295.660,A 0.000,B 0.000,C 90.000,E1 154.845} C_DIS
LIN {X -0.185,Y -500.801,Z 1295.659,A 0.000,B 0.000,C 90.000,E1 154.588} C_DIS
LIN {X 0.118,Y -504.077,Z 1295.657,A 0.000,B 0.000,C 90.000,E1 154.229} C_DIS
LIN {X 0.192,Y -510.392,Z 1295.653,A 0.000,B 0.000,C 90.000,E1 153.512} C_DIS
LIN {X -0.061,Y -515.397,Z 1295.650,A 0.000,B 0.000,C 90.000,E1 152.948} C_DIS
LIN {X -0.051,Y -519.927,Z 1295.646,A 0.000,B 0.000,C 90.000,E1 152.359} C_DIS
LIN {X 0.159,Y -523.160,Z 1295.644,A 0.000,B 0.000,C 90.000,E1 151.897} C_DIS
LIN {X 0.233,Y -526.955,Z 1295.641,A 0.000,B 0.000,C 90.000,E1 151.307} C_DIS
LIN {X 0.184,Y -530.973,Z 1295.637,A 0.000,B 0.000,C 90.000,E1 150.589} C_DIS
LIN {X -0.147,Y -533.775,Z 1295.634,A 0.000,B 0.000,C 90.000,E1 150.049} C_DIS
LIN {X 0.023,Y -534.905,Z 1295.632,A 0.000,B 0.000,C 90.000,E1 149.744} C_DIS
LIN {X 0.003,Y -536.504,Z 1295.630,A 0.000,B 0.000,C 90.000,E1 149.459} C_DIS
LIN {X 0.178,Y -538.050,Z 1295.629,A 0.000,B 0.000,C 90.000,E1 149.203} C_DIS
LIN {X 0.036,Y -538.805,Z 1295.628,A 0.000,B 0.000,C 90.000,E1 149.076} C_DIS
LIN {X -0.106,Y -539.368,Z 1295.627,A 0.000,B 0.000,C 90.000,E1 148.948} C_DIS
LIN {X 0.033,Y -540.288,Z 1295.627,A 0.000,B 0.000,C 90.000,E1 148.791} C_DIS
LIN {X -0.106,Y -541.600,Z 1295.626,A 0.000,B 0.000,C 90.000,E1 148.663} C_DIS
LIN {X -0.251,Y -548.104,Z 1295.623,A 0.000,B 0.000,C 90.000,E1 148.201} C_DIS
LIN {X 0.124,Y -561.740,Z 1295.618,A 0.000,B 0.000,C 90.000,E1 147.248} C_DIS
LIN {X 0.164,Y -568.960,Z 1295.615,A 0.000,B 0.000,C 90.000,E1 146.707} C_DIS
LIN {X 0.048,Y -576.390,Z 1295.612,A 0.000,B 0.000,C 90.000,E1 146.167} C_DIS
LIN {X -0.005,Y -581.940,Z 1295.610,A 0.000,B 0.000,C 90.000,E1 145.722} C_DIS
LIN {X -0.089,Y -590.238,Z 1295.606,A 0.000,B 0.000,C 90.000,E1 145.022} C_DIS
LIN {X 0.123,Y -594.047,Z 1295.604,A 0.000,B 0.000,C 90.000,E1 144.642} C_DIS
LIN {X 0.277,Y -600.295,Z 1295.600,A 0.000,B 0.000,C 90.000,E1 143.989} C_DIS
LIN {X 0.006,Y -603.813,Z 1295.598,A 0.000,B 0.000,C 90.000,E1 143.623} C_DIS
LIN {X 0.213,Y -607.108,Z 1295.596,A 0.000,B 0.000,C 90.000,E1 143.210} C_DIS
LIN {X 0.229,Y -612.050,Z 1295.592,A 0.000,B 0.000,C 90.000,E1 142.557} C_DIS
LIN {X -0.009,Y -614.832,Z 1295.590,A 0.000,B 0.000,C 90.000,E1 142.190} C_DIS
LIN {X 0.110,Y -618.288,Z 1295.587,A 0.000,B 0.000,C 90.000,E1 141.662} C_DIS
LIN {X -0.326,Y -623.966,Z 1295.582,A 0.000,B 0.000,C 90.000,E1 140.803} C_DIS
LIN {X -0.170,Y -627.587,Z 1295.579,A 0.000,B 0.000,C 90.000,E1 140.150} C_DIS
LIN {X 0.040,Y -630.325,Z 1295.576,A 0.000,B 0.000,C 90.000,E1 139.622} C_DIS
LIN {X -0.349,Y -634.779,Z 1295.571,A 0.000,B 0.000,C 90.000,E1 138.771} C_DIS
LIN {X -0.191,Y -638.234,Z 1295.567,A 0.000,B 0.000,C 90.000,E1 138.000} C_DIS
LIN {X -0.083,Y -642.650,Z 1295.561,A 0.000,B 0.000,C 90.000,E1 136.986} C_DIS
LIN {X -0.047,Y -648.938,Z 1295.553,A 0.000,B 0.000,C 90.000,E1 135.486} C_DIS
LIN {X -0.312,Y -654.028,Z 1295.546,A 0.000,B 0.000,C 90.000,E1 134.271} C_DIS
LIN {X -0.025,Y -659.012,Z 1295.539,A 0.000,B 0.000,C 90.000,E1 133.014} C_DIS
LIN {X 0.350,Y -663.946,Z 1295.532,A 0.000,B 0.000,C 90.000,E1 131.757} C_DIS
LIN {X -0.120,Y -665.887,Z 1295.530,A 0.000,B 0.000,C 90.000,E1 131.310} C_DIS
LIN {X -0.081,Y -670.446,Z 1295.523,A 0.000,B 0.000,C 90.000,E1 130.092} C_DIS
LIN {X 0.022,Y -674.668,Z 1295.516,A 0.000,B 0.000,C 90.000,E1 128.874} C_DIS
LIN {X 0.290,Y -678.600,Z 1295.509,A 0.000,B 0.000,C 90.000,E1 127.649} C_DIS
LIN {X 0.065,Y -681.458,Z 1295.504,A 0.000,B 0.000,C 90.000,E1 126.710} C_DIS
LIN {X 0.024,Y -684.120,Z 1295.499,A 0.000,B 0.000,C 90.000,E1 125.758} C_DIS
LIN {X -0.135,Y -686.598,Z 1295.493,A 0.000,B 0.000,C 90.000,E1 124.818} C_DIS
LIN {X -0.296,Y -688.294,Z 1295.490,A 0.000,B 0.000,C 90.000,E1 124.119} C_DIS
LIN {X -0.232,Y -690.312,Z 1295.484,A 0.000,B 0.000,C 90.000,E1 123.166} C_DIS
LIN {X -0.140,Y -692.062,Z 1295.479,A 0.000,B 0.000,C 90.000,E1 122.212} C_DIS
LIN {X -0.029,Y -693.583,Z 1295.474,A 0.000,B 0.000,C 90.000,E1 121.258} C_DIS
LIN {X -0.365,Y -695.766,Z 1295.466,A 0.000,B 0.000,C 90.000,E1 119.873} C_DIS
LIN {X 0.045,Y -697.005,Z 1295.461,A 0.000,B 0.000,C 90.000,E1 118.899} C_DIS
LIN {X -0.401,Y -697.752,Z 1295.457,A 0.000,B 0.000,C 90.000,E1 118.231} C_DIS
LIN {X -0.231,Y -698.275,Z 1295.453,A 0.000,B 0.000,C 90.000,E1 117.513} C_DIS
LIN {X -0.059,Y -698.569,Z 1295.449,A 0.000,B 0.000,C 90.000,E1 116.796} C_DIS
LIN {X -0.198,Y -698.656,Z 1295.445,A 0.000,B 0.000,C 90.000,E1 116.104} C_DIS
LIN {X -0.332,Y -698.385,Z 1295.441,A 0.000,B 0.000,C 90.000,E1 115.412} C_DIS
LIN {X 0.199,Y -698.000,Z 1295.438,A 0.000,B 0.000,C 90.000,E1 114.899} C_DIS
LIN {X -0.200,Y -697.254,Z 1295.436,A 0.000,B 0.000,C 90.000,E1 114.463} C_DIS
LIN {X 0.061,Y -696.801,Z 1295.435,A 0.000,B 0.000,C 90.000,E1 114.207} C_DIS
LIN {X -0.343,Y -695.202,Z 1295.432,A 0.000,B 0.000,C 90.000,E1 113.770} C_DIS
LIN {X -0.089,Y -694.028,Z 1295.431,A 0.000,B 0.000,C 90.000,E1 113.515} C_DIS
LIN {X 0.127,Y -690.723,Z 1295.428,A 0.000,B 0.000,C 90.000,E1 113.025} C_DIS
LIN {X 0.246,Y -689.516,Z 1295.427,A 0.000,B 0.000,C 90.000,E1 112.898} C_DIS
LIN {X 0.002,Y -683.395,Z 1295.425,A 0.000,B 0.000,C 90.000,E1 112.514} C_DIS
LIN {X 0.131,Y -681.668,Z 1295.425,A 0.000,B 0.000,C 90.000,E1 112.408} C_DIS
LIN {X 0.011,Y -679.050,Z 1295.424,A 0.000,B 0.000,C 90.000,E1 112.333} C_DIS
LIN {X 0.061,Y -672.306,Z 1295.423,A 0.000,B 0.000,C 90.000,E1 112.153} C_DIS
LIN {X 0.140,Y -669.432,Z 1295.423,A 0.000,B 0.000,C 90.000,E1 112.099} C_DIS
LIN {X 0.241,Y -662.471,Z 1295.422,A 0.000,B 0.000,C 90.000,E1 112.025} C_DIS
LIN {X 0.182,Y -655.785,Z 1295.422,A 0.000,B 0.000,C 90.000,E1 112.025} C_DIS
LIN {X 0.126,Y -648.917,Z 1295.422,A 0.000,B 0.000,C 90.000,E1 112.025} C_DIS
LIN {X -0.148,Y -644.776,Z 1295.422,A 0.000,B 0.000,C 90.000,E1 112.025} C_DIS
LIN {X 0.021,Y -642.552,Z 1295.422,A 0.000,B 0.000,C 90.000,E1 111.972} C_DIS
LIN {X -0.072,Y -639.738,Z 1295.422,A 0.000,B 0.000,C 90.000,E1 111.897} C_DIS
LIN {X -0.109,Y -639.729,Z 1295.422,A 0.000,B 0.000,C 90.000,E1 111.897} C_DIS
LIN {X -0.171,Y -641.257,Z 1295.420,A 0.000,B 0.000,C 90.000,E1 111.589} C_DIS
LIN {X -0.181,Y -642.399,Z 1295.419,A 0.000,B 0.000,C 90.000,E1 111.408} C_DIS
LIN {X 0.185,Y -649.634,Z 1295.414,A 0.000,B 0.000,C 90.000,E1 110.429} C_DIS
LIN {X 0.076,Y -652.160,Z 1295.412,A 0.000,B 0.000,C 90.000,E1 110.066} C_DIS
LIN {X 0.024,Y -655.335,Z 1295.409,A 0.000,B 0.000,C 90.000,E1 109.577} C_DIS
LIN {X -0.079,Y -660.030,Z 1295.404,A 0.000,B 0.000,C 90.000,E1 108.725} C_DIS
LIN {X -0.190,Y -663.489,Z 1295.400,A 0.000,B 0.000,C 90.000,E1 108.000} C_DIS
LIN {X -0.273,Y -666.484,Z 1295.396,A 0.000,B 0.000,C 90.000,E1 107.275} C_DIS
LIN {X 0.197,Y -668.294,Z 1295.393,A 0.000,B 0.000,C 90.000,E1 106.749} C_DIS
LIN {X 0.162,Y -670.608,Z 1295.389,A 0.000,B 0.000,C 90.000,E1 106.024} C_DIS
LIN {X 0.140,Y -672.470,Z 1295.385,A 0.000,B 0.000,C 90.000,E1 105.300} C_DIS
LIN {X -0.046,Y -674.081,Z 1295.381,A 0.000,B 0.000,C 90.000,E1 104.592} C_DIS
LIN {X -0.160,Y -674.913,Z 1295.378,A 0.000,B 0.000,C 90.000,E1 104.120} C_DIS
LIN {X 0.337,Y -675.966,Z 1295.374,A 0.000,B 0.000,C 90.000,E1 103.355} C_DIS
LIN {X 0.186,Y -676.594,Z 1295.370,A 0.000,B 0.000,C 90.000,E1 102.647} C_DIS
LIN {X -0.104,Y -676.847,Z 1295.366,A 0.000,B 0.000,C 90.000,E1 101.951} C_DIS
LIN {X -0.201,Y -676.800,Z 1295.364,A 0.000,B 0.000,C 90.000,E1 101.478} C_DIS
LIN {X 0.362,Y -676.565,Z 1295.361,A 0.000,B 0.000,C 90.000,E1 100.950} C_DIS
LIN {X 0.079,Y -675.837,Z 1295.357,A 0.000,B 0.000,C 90.000,E1 100.254} C_DIS
LIN {X -0.150,Y -675.086,Z 1295.354,A 0.000,B 0.000,C 90.000,E1 99.792} C_DIS
LIN {X -0.269,Y -674.062,Z 1295.352,A 0.000,B 0.000,C 90.000,E1 99.321} C_DIS
LIN {X 0.161,Y -672.688,Z 1295.349,A 0.000,B 0.000,C 90.000,E1 98.803} C_DIS
LIN {X -0.081,Y -671.024,Z 1295.346,A 0.000,B 0.000,C 90.000,E1 98.341} C_DIS
LIN {X -0.236,Y -669.006,Z 1295.344,A 0.000,B 0.000,C 90.000,E1 97.871} C_DIS
LIN {X 0.162,Y -666.691,Z 1295.341,A 0.000,B 0.000,C 90.000,E1 97.352} C_DIS
LIN {X -0.024,Y -664.803,Z 1295.339,A 0.000,B 0.000,C 90.000,E1 97.004} C_DIS
LIN {X 0.247,Y -661.254,Z 1295.336,A 0.000,B 0.000,C 90.000,E1 96.372} C_DIS
LIN {X -0.067,Y -658.210,Z 1295.333,A 0.000,B 0.000,C 90.000,E1 95.910} C_DIS
LIN {X 0.251,Y -654.780,Z 1295.330,A 0.000,B 0.000,C 90.000,E1 95.391} C_DIS
LIN {X -0.268,Y -650.058,Z 1295.327,A 0.000,B 0.000,C 90.000,E1 94.821} C_DIS
LIN {X 0.108,Y -647.049,Z 1295.325,A 0.000,B 0.000,C 90.000,E1 94.416} C_DIS
LIN {X 0.108,Y -640.263,Z 1295.320,A 0.000,B 0.000,C 90.000,E1 93.669} C_DIS
LIN {X 0.106,Y -633.016,Z 1295.316,A 0.000,B 0.000,C 90.000,E1 92.922} C_DIS
LIN {X 0.134,Y -625.663,Z 1295.312,A 0.000,B 0.000,C 90.000,E1 92.178} C_DIS
LIN {X -0.153,Y -620.435,Z 1295.310,A 0.000,B 0.000,C 90.000,E1 91.718} C_DIS
LIN {X -0.271,Y -616.225,Z 1295.307,A 0.000,B 0.000,C 90.000,E1 91.375} C_DIS
LIN {X 0.277,Y -608.996,Z 1295.305,A 0.000,B 0.000,C 90.000,E1 90.802} C_DIS
LIN {X 0.218,Y -602.580,Z 1295.302,A 0.000,B 0.000,C 90.000,E1 90.401} C_DIS
LIN {X -0.024,Y -596.006,Z 1295.300,A 0.000,B 0.000,C 90.000,E1 90.057} C_DIS
LIN {X 0.109,Y -589.041,Z 1295.298,A 0.000,B 0.000,C 90.000,E1 89.714} C_DIS
LIN {X 0.088,Y -581.441,Z 1295.297,A 0.000,B 0.000,C 90.000,E1 89.427} C_DIS
LIN {X -0.036,Y -576.223,Z 1295.296,A 0.000,B 0.000,C 90.000,E1 89.255} C_DIS
LIN {X -0.239,Y -572.211,Z 1295.295,A 0.000,B 0.000,C 90.000,E1 89.083} C_DIS
LIN {X -0.243,Y -570.188,Z 1295.294,A 0.000,B 0.000,C 90.000,E1 88.912} C_DIS
LIN {X -0.282,Y -570.171,Z 1295.294,A 0.000,B 0.000,C 90.000,E1 88.912} C_DIS
LIN {X -0.179,Y -569.870,Z 1295.293,A 0.000,B 0.000,C 90.000,E1 88.797} C_DIS
LIN {X 0.091,Y -569.737,Z 1295.292,A 0.000,B 0.000,C 90.000,E1 88.511} C_DIS
LIN {X 0.217,Y -569.705,Z 1295.290,A 0.000,B 0.000,C 90.000,E1 88.224} C_DIS
LIN {X 0.002,Y -572.208,Z 1295.274,A 0.000,B 0.000,C 90.000,E1 85.241} C_DIS
LIN {X -0.025,Y -574.326,Z 1295.263,A 0.000,B 0.000,C 90.000,E1 83.337} C_DIS
LIN {X 0.214,Y -576.887,Z 1295.251,A 0.000,B 0.000,C 90.000,E1 81.141} C_DIS
LIN {X 0.268,Y -578.791,Z 1295.242,A 0.000,B 0.000,C 90.000,E1 79.511} C_DIS
LIN {X -0.094,Y -579.892,Z 1295.236,A 0.000,B 0.000,C 90.000,E1 78.465} C_DIS
LIN {X -0.102,Y -581.122,Z 1295.228,A 0.000,B 0.000,C 90.000,E1 77.117} C_DIS
LIN {X -0.183,Y -582.056,Z 1295.222,A 0.000,B 0.000,C 90.000,E1 76.047} C_DIS
LIN {X 0.220,Y -583.267,Z 1295.214,A 0.000,B 0.000,C 90.000,E1 74.393} C_DIS
LIN {X -0.095,Y -584.503,Z 1295.203,A 0.000,B 0.000,C 90.000,E1 72.543} C_DIS
LIN {X 0.122,Y -585.553,Z 1295.194,A 0.000,B 0.000,C 90.000,E1 70.913} C_DIS
LIN {X 0.088,Y -586.848,Z 1295.182,A 0.000,B 0.000,C 90.000,E1 68.773} C_DIS
LIN {X -0.242,Y -588.132,Z 1295.170,A 0.000,B 0.000,C 90.000,E1 66.666} C_DIS
LIN {X -0.088,Y -589.293,Z 1295.161,A 0.000,B 0.000,C 90.000,E1 65.049} C_DIS
LIN {X 0.058,Y -590.454,Z 1295.152,A 0.000,B 0.000,C 90.000,E1 63.435} C_DIS
LIN {X 0.144,Y -592.019,Z 1295.142,A 0.000,B 0.000,C 90.000,E1 61.563} C_DIS
LIN {X -0.166,Y -593.602,Z 1295.133,A 0.000,B 0.000,C 90.000,E1 59.999} C_DIS
LIN {X 0.042,Y -594.697,Z 1295.127,A 0.000,B 0.000,C 90.000,E1 58.918} C_DIS
LIN {X 0.174,Y -596.025,Z 1295.120,A 0.000,B 0.000,C 90.000,E1 57.582} C_DIS
LIN {X -0.184,Y -597.447,Z 1295.113,A 0.000,B 0.000,C 90.000,E1 56.294} C_DIS
LIN {X -0.191,Y -598.821,Z 1295.105,A 0.000,B 0.000,C 90.000,E1 54.975} C_DIS
LIN {X 0.059,Y -600.279,Z 1295.097,A 0.000,B 0.000,C 90.000,E1 53.371} C_DIS
LIN {X -0.262,Y -601.585,Z 1295.088,A 0.000,B 0.000,C 90.000,E1 51.823} C_DIS
LIN {X 0.016,Y -602.283,Z 1295.083,A 0.000,B 0.000,C 90.000,E1 51.009} C_DIS
LIN {X -0.046,Y -603.077,Z 1295.076,A 0.000,B 0.000,C 90.000,E1 49.703} C_DIS
LIN {X 0.033,Y -603.615,Z 1295.070,A 0.000,B 0.000,C 90.000,E1 48.647} C_DIS
LIN {X -0.130,Y -603.849,Z 1295.066,A 0.000,B 0.000,C 90.000,E1 47.877} C_DIS
LIN {X -0.036,Y -604.295,Z 1295.057,A 0.000,B 0.000,C 90.000,E1 46.296} C_DIS
LIN {X 0.030,Y -604.387,Z 1295.051,A 0.000,B 0.000,C 90.000,E1 45.243} C_DIS
LIN {X 0.099,Y -604.345,Z 1295.046,A 0.000,B 0.000,C 90.000,E1 44.190} C_DIS
LIN {X -0.039,Y -603.998,Z 1295.038,A 0.000,B 0.000,C 90.000,E1 42.894} C_DIS
LIN {X 0.048,Y -603.721,Z 1295.032,A 0.000,B 0.000,C 90.000,E1 41.838} C_DIS
LIN {X -0.110,Y -603.400,Z 1295.028,A 0.000,B 0.000,C 90.000,E1 41.067} C_DIS
LIN {X 0.265,Y -602.556,Z 1295.018,A 0.000,B 0.000,C 90.000,E1 39.197} C_DIS
LIN {X -0.043,Y -601.873,Z 1295.012,A 0.000,B 0.000,C 90.000,E1 38.177} C_DIS
LIN {X -0.359,Y -600.956,Z 1295.006,A 0.000,B 0.000,C 90.000,E1 37.156} C_DIS
LIN {X -0.210,Y -599.722,Z 1295.000,A 0.000,B 0.000,C 90.000,E1 36.091} C_DIS
LIN {X -0.079,Y -598.290,Z 1294.995,A 0.000,B 0.000,C 90.000,E1 35.025} C_DIS
LIN {X -0.084,Y -595.947,Z 1294.987,A 0.000,B 0.000,C 90.000,E1 33.706} C_DIS
LIN {X 0.256,Y -594.381,Z 1294.983,A 0.000,B 0.000,C 90.000,E1 32.880} C_DIS
LIN {X 0.364,Y -593.191,Z 1294.980,A 0.000,B 0.000,C 90.000,E1 32.339} C_DIS
LIN {X -0.147,Y -591.048,Z 1294.975,A 0.000,B 0.000,C 90.000,E1 31.592} C_DIS
LIN {X 0.013,Y -587.835,Z 1294.970,A 0.000,B 0.000,C 90.000,E1 30.512} C_DIS
LIN {X -0.051,Y -584.832,Z 1294.965,A 0.000,B 0.000,C 90.000,E1 29.716} C_DIS
LIN {X 0.209,Y -582.668,Z 1294.962,A 0.000,B 0.000,C 90.000,E1 29.155} C_DIS
LIN {X 0.027,Y -578.450,Z 1294.957,A 0.000,B 0.000,C 90.000,E1 28.231} C_DIS
LIN {X -0.065,Y -574.984,Z 1294.953,A 0.000,B 0.000,C 90.000,E1 27.564} C_DIS
LIN {X 0.054,Y -571.150,Z 1294.949,A 0.000,B 0.000,C 90.000,E1 26.873} C_DIS
LIN {X -0.278,Y -567.911,Z 1294.946,A 0.000,B 0.000,C 90.000,E1 26.360} C_DIS
LIN {X -0.062,Y -562.675,Z 1294.942,A 0.000,B 0.000,C 90.000,E1 25.515} C_DIS
LIN {X -0.150,Y -556.817,Z 1294.937,A 0.000,B 0.000,C 90.000,E1 24.695} C_DIS
LIN {X -0.075,Y -552.619,Z 1294.934,A 0.000,B 0.000,C 90.000,E1 24.131} C_DIS
LIN {X -0.028,Y -548.101,Z 1294.931,A 0.000,B 0.000,C 90.000,E1 23.567} C_DIS
LIN {X -0.111,Y -539.659,Z 1294.926,A 0.000,B 0.000,C 90.000,E1 22.589} C_DIS
LIN {X -0.156,Y -534.630,Z 1294.922,A 0.000,B 0.000,C 90.000,E1 22.025} C_DIS
LIN {X -0.147,Y -525.553,Z 1294.917,A 0.000,B 0.000,C 90.000,E1 21.046} C_DIS
LIN {X 0.251,Y -518.889,Z 1294.913,A 0.000,B 0.000,C 90.000,E1 20.301} C_DIS
LIN {X 0.039,Y -512.129,Z 1294.909,A 0.000,B 0.000,C 90.000,E1 19.631} C_DIS
LIN {X 0.292,Y -503.870,Z 1294.905,A 0.000,B 0.000,C 90.000,E1 18.779} C_DIS
LIN {X -0.162,Y -494.136,Z 1294.899,A 0.000,B 0.000,C 90.000,E1 17.873} C_DIS
LIN {X 0.106,Y -484.355,Z 1294.894,A 0.000,B 0.000,C 90.000,E1 16.913} C_DIS
LIN {X -0.263,Y -474.007,Z 1294.889,A 0.000,B 0.000,C 90.000,E1 16.024} C_DIS
LIN {X -0.029,Y -463.671,Z 1294.884,A 0.000,B 0.000,C 90.000,E1 15.064} C_DIS
LIN {X -0.022,Y -449.071,Z 1294.876,A 0.000,B 0.000,C 90.000,E1 13.716} C_DIS
LIN {X -0.137,Y -425.927,Z 1294.863,A 0.000,B 0.000,C 90.000,E1 11.422} C_DIS
LIN {X 0.157,Y -407.305,Z 1294.852,A 0.000,B 0.000,C 90.000,E1 9.378} C_DIS
LIN {X -0.078,Y -400.339,Z 1294.848,A 0.000,B 0.000,C 90.000,E1 8.624} C_DIS
LIN {X 0.100,Y -396.532,Z 1294.845,A 0.000,B 0.000,C 90.000,E1 8.106} C_DIS
LIN {X -0.080,Y -395.225,Z 1294.844,A 0.000,B 0.000,C 90.000,E1 7.871} C_DIS
LIN {X -0.117,Y -395.250,Z 1294.844,A 0.000,B 0.000,C 90.000,E1 7.871} C_DIS
LIN {X -0.083,Y -396.284,Z 1294.843,A 0.000,B 0.000,C 90.000,E1 7.701} C_DIS
LIN {X -0.062,Y -398.799,Z 1294.841,A 0.000,B 0.000,C 90.000,E1 7.466} C_DIS
LIN {X 0.125,Y -400.581,Z 1294.841,A 0.000,B 0.000,C 90.000,E1 7.296} C_DIS
LIN {X 0.083,Y -406.515,Z 1294.839,A 0.000,B 0.000,C 90.000,E1 6.947} C_DIS
LIN {X 0.089,Y -409.616,Z 1294.838,A 0.000,B 0.000,C 90.000,E1 6.777} C_DIS
LIN {X 0.166,Y -415.796,Z 1294.836,A 0.000,B 0.000,C 90.000,E1 6.372} C_DIS
LIN {X -0.142,Y -423.932,Z 1294.833,A 0.000,B 0.000,C 90.000,E1 5.853} C_DIS
LIN {X 0.117,Y -431.687,Z 1294.829,A 0.000,B 0.000,C 90.000,E1 5.220} C_DIS
LIN {X -0.198,Y -437.898,Z 1294.826,A 0.000,B 0.000,C 90.000,E1 4.759} C_DIS
LIN {X -0.035,Y -447.121,Z 1294.822,A 0.000,B 0.000,C 90.000,E1 3.955} C_DIS
LIN {X 0.161,Y -454.578,Z 1294.818,A 0.000,B 0.000,C 90.000,E1 3.269} C_DIS
LIN {X 0.143,Y -461.717,Z 1294.814,A 0.000,B 0.000,C 90.000,E1 2.579} C_DIS
LIN {X 0.119,Y -467.363,Z 1294.811,A 0.000,B 0.000,C 90.000,E1 2.007} C_DIS
LIN {X -0.045,Y -472.834,Z 1294.808,A 0.000,B 0.000,C 90.000,E1 1.432} C_DIS
LIN {X 0.125,Y -477.848,Z 1294.805,A 0.000,B 0.000,C 90.000,E1 0.802} C_DIS
LIN {X 0.207,Y -482.756,Z 1294.801,A 0.000,B 0.000,C 90.000,E1 0.172} C_DIS
LIN {X 0.006,Y -487.970,Z 1294.797,A 0.000,B 0.000,C 90.000,E1 359.484} C_DIS
LIN {X 0.008,Y -494.019,Z 1294.792,A 0.000,B 0.000,C 90.000,E1 358.568} C_DIS
LIN {X 0.229,Y -497.896,Z 1294.789,A 0.000,B 0.000,C 90.000,E1 357.936} C_DIS
LIN {X -0.162,Y -503.082,Z 1294.784,A 0.000,B 0.000,C 90.000,E1 357.078} C_DIS
LIN {X 0.136,Y -506.400,Z 1294.780,A 0.000,B 0.000,C 90.000,E1 356.445} C_DIS
LIN {X 0.164,Y -510.271,Z 1294.776,A 0.000,B 0.000,C 90.000,E1 355.698} C_DIS
LIN {X 0.226,Y -513.897,Z 1294.772,A 0.000,B 0.000,C 90.000,E1 354.951} C_DIS
LIN {X 0.105,Y -516.663,Z 1294.769,A 0.000,B 0.000,C 90.000,E1 354.375} C_DIS
LIN {X 0.002,Y -519.228,Z 1294.766,A 0.000,B 0.000,C 90.000,E1 353.799} C_DIS
LIN {X -0.090,Y -522.795,Z 1294.761,A 0.000,B 0.000,C 90.000,E1 352.932} C_DIS
LIN {X -0.146,Y -526.088,Z 1294.756,A 0.000,B 0.000,C 90.000,E1 352.064} C_DIS
LIN {X -0.190,Y -528.092,Z 1294.753,A 0.000,B 0.000,C 90.000,E1 351.489} C_DIS
LIN {X -0.163,Y -531.764,Z 1294.746,A 0.000,B 0.000,C 90.000,E1 350.330} C_DIS
LIN {X -0.038,Y -534.250,Z 1294.741,A 0.000,B 0.000,C 90.000,E1 349.454} C_DIS
LIN {X 0.119,Y -536.493,Z 1294.737,A 0.000,B 0.000,C 90.000,E1 348.578} C_DIS
LIN {X -0.226,Y -538.537,Z 1294.732,A 0.000,B 0.000,C 90.000,E1 347.757} C_DIS
LIN {X -0.026,Y -540.306,Z 1294.727,A 0.000,B 0.000,C 90.000,E1 346.881} C_DIS
LIN {X -0.207,Y -541.865,Z 1294.722,A 0.000,B 0.000,C 90.000,E1 346.047} C_DIS
LIN {X 0.022,Y -543.220,Z 1294.718,A 0.000,B 0.000,C 90.000,E1 345.172} C_DIS
LIN {X 0.102,Y -544.638,Z 1294.711,A 0.000,B 0.000,C 90.000,E1 344.031} C_DIS
LIN {X 0.054,Y -545.639,Z 1294.705,A 0.000,B 0.000,C 90.000,E1 342.906} C_DIS
LIN {X 0.096,Y -546.141,Z 1294.700,A 0.000,B 0.000,C 90.000,E1 342.054} C_DIS
LIN {X -0.025,Y -546.362,Z 1294.696,A 0.000,B 0.000,C 90.000,E1 341.221} C_DIS
LIN {X 0.028,Y -546.237,Z 1294.691,A 0.000,B 0.000,C 90.000,E1 340.369} C_DIS
LIN {X 0.080,Y -545.839,Z 1294.686,A 0.000,B 0.000,C 90.000,E1 339.518} C_DIS
LIN {X 0.124,Y -545.111,Z 1294.682,A 0.000,B 0.000,C 90.000,E1 338.666} C_DIS
LIN {X 0.113,Y -544.471,Z 1294.678,A 0.000,B 0.000,C 90.000,E1 338.103} C_DIS
LIN {X 0.325,Y -542.295,Z 1294.671,A 0.000,B 0.000,C 90.000,E1 336.666} C_DIS
LIN {X 0.065,Y -541.651,Z 1294.669,A 0.000,B 0.000,C 90.000,E1 336.410} C_DIS
LIN {X 0.301,Y -541.238,Z 1294.667,A 0.000,B 0.000,C 90.000,E1 336.102} C_DIS
LIN {X 0.006,Y -539.078,Z 1294.663,A 0.000,B 0.000,C 90.000,E1 335.281} C_DIS
LIN {X 0.173,Y -536.689,Z 1294.658,A 0.000,B 0.000,C 90.000,E1 334.409} C_DIS
LIN {X -0.023,Y -532.117,Z 1294.650,A 0.000,B 0.000,C 90.000,E1 332.999} C_DIS
LIN {X -0.175,Y -529.328,Z 1294.645,A 0.000,B 0.000,C 90.000,E1 332.153} C_DIS
LIN {X 0.109,Y -526.196,Z 1294.640,A 0.000,B 0.000,C 90.000,E1 331.257} C_DIS
LIN {X 0.205,Y -523.824,Z 1294.637,A 0.000,B 0.000,C 90.000,E1 330.667} C_DIS
LIN {X 0.116,Y -520.591,Z 1294.633,A 0.000,B 0.000,C 90.000,E1 329.950} C_DIS
LIN {X 0.089,Y -516.327,Z 1294.628,A 0.000,B 0.000,C 90.000,E1 329.076} C_DIS
LIN {X 0.198,Y -512.602,Z 1294.624,A 0.000,B 0.000,C 90.000,E1 328.329} C_DIS
LIN {X 0.311,Y -505.270,Z 1294.616,A 0.000,B 0.000,C 90.000,E1 326.834} C_DIS
LIN {X -0.060,Y -502.772,Z 1294.613,A 0.000,B 0.000,C 90.000,E1 326.294} C_DIS
LIN {X -0.079,Y -500.687,Z 1294.610,A 0.000,B 0.000,C 90.000,E1 325.722} C_DIS
LIN {X -0.032,Y -498.246,Z 1294.605,A 0.000,B 0.000,C 90.000,E1 324.815} C_DIS
LIN {X -0.013,Y -496.645,Z 1294.599,A 0.000,B 0.000,C 90.000,E1 323.909} C_DIS
LIN {X 0.006,Y -495.193,Z 1294.591,A 0.000,B 0.000,C 90.000,E1 322.396} C_DIS
LIN {X 0.140,Y -494.686,Z 1294.584,A 0.000,B 0.000,C 90.000,E1 321.170} C_DIS
LIN {X -0.038,Y -494.807,Z 1294.568,A 0.000,B 0.000,C 90.000,E1 318.162} C_DIS
LIN {X 0.199,Y -494.985,Z 1294.559,A 0.000,B 0.000,C 90.000,E1 316.620} C_DIS
LIN {X 0.072,Y -495.154,Z 1294.551,A 0.000,B 0.000,C 90.000,E1 315.121} C_DIS
LIN {X 0.277,Y -495.133,Z 1294.546,A 0.000,B 0.000,C 90.000,E1 314.190} C_DIS
LIN {X -0.053,Y -494.930,Z 1294.542,A 0.000,B 0.000,C 90.000,E1 313.623} C_DIS
LIN {X 0.156,Y -494.206,Z 1294.537,A 0.000,B 0.000,C 90.000,E1 312.690} C_DIS
LIN {X 0.003,Y -493.841,Z 1294.536,A 0.000,B 0.000,C 90.000,E1 312.405} C_DIS
LIN {X 0.182,Y -493.345,Z 1294.534,A 0.000,B 0.000,C 90.000,E1 312.081} C_DIS
LIN {X -0.338,Y -492.692,Z 1294.532,A 0.000,B 0.000,C 90.000,E1 311.838} C_DIS
LIN {X -0.165,Y -491.790,Z 1294.531,A 0.000,B 0.000,C 90.000,E1 311.515} C_DIS
LIN {X -0.082,Y -491.159,Z 1294.530,A 0.000,B 0.000,C 90.000,E1 311.353} C_DIS
LIN {X 0.003,Y -490.248,Z 1294.529,A 0.000,B 0.000,C 90.000,E1 311.191} C_DIS
LIN {X -0.127,Y -471.575,Z 1294.514,A 0.000,B 0.000,C 90.000,E1 308.588} C_DIS
LIN {X -0.001,Y -454.777,Z 1294.499,A 0.000,B 0.000,C 90.000,E1 305.884} C_DIS
LIN {X -0.285,Y -439.734,Z 1294.484,A 0.000,B 0.000,C 90.000,E1 303.166} C_DIS
LIN {X -0.176,Y -426.341,Z 1294.469,A 0.000,B 0.000,C 90.000,E1 300.335} C_DIS
LIN {X 0.000,Y -414.500,Z 1294.453,A 0.000,B 0.000,C 90.000,E1 297.436} C_DIS
LIN {X -0.042,Y -404.136,Z 1294.436,A 0.000,B 0.000,C 90.000,E1 294.515} C_DIS
LIN {X -0.054,Y -400.782,Z 1294.430,A 0.000,B 0.000,C 90.000,E1 293.462} C_DIS
LIN {X -0.093,Y -400.785,Z 1294.430,A 0.000,B 0.000,C 90.000,E1 293.462} C_DIS
LIN {X -0.026,Y -401.542,Z 1294.427,A 0.000,B 0.000,C 90.000,E1 292.770} C_DIS
LIN {X -0.154,Y -402.622,Z 1294.411,A 0.000,B 0.000,C 90.000,E1 289.993} C_DIS
LIN {X 0.115,Y -404.608,Z 1294.396,A 0.000,B 0.000,C 90.000,E1 287.166} C_DIS
LIN {X -0.170,Y -404.756,Z 1294.394,A 0.000,B 0.000,C 90.000,E1 286.858} C_DIS
LIN {X 0.217,Y -406.067,Z 1294.365,A 0.000,B 0.000,C 90.000,E1 281.591} C_DIS
LIN {X -0.174,Y -406.118,Z 1294.363,A 0.000,B 0.000,C 90.000,E1 281.299} C_DIS
LIN {X -0.143,Y -405.667,Z 1294.334,A 0.000,B 0.000,C 90.000,E1 276.087} C_DIS
LIN {X -0.139,Y -405.566,Z 1294.332,A 0.000,B 0.000,C 90.000,E1 275.739} C_DIS
LIN {X -0.064,Y -403.530,Z 1294.305,A 0.000,B 0.000,C 90.000,E1 270.859} C_DIS
LIN {X -0.129,Y -402.987,Z 1294.301,A 0.000,B 0.000,C 90.000,E1 270.172} C_DIS
LIN {X 0.091,Y -398.981,Z 1294.272,A 0.000,B 0.000,C 90.000,E1 264.894} C_DIS
LIN {X -0.103,Y -393.153,Z 1294.242,A 0.000,B 0.000,C 90.000,E1 259.634} C_DIS
LIN {X -0.071,Y -392.888,Z 1294.240,A 0.000,B 0.000,C 90.000,E1 259.275} C_DIS
LIN {X 0.113,Y -389.618,Z 1294.229,A 0.000,B 0.000,C 90.000,E1 257.117} C_DIS
LIN {X -0.003,Y -385.324,Z 1294.209,A 0.000,B 0.000,C 90.000,E1 253.559} C_DIS
LIN {X 0.003,Y -384.667,Z 1294.206,A 0.000,B 0.000,C 90.000,E1 253.087} C_DIS
LIN {X -0.035,Y -384.676,Z 1294.206,A 0.000,B 0.000,C 90.000,E1 253.087} C_DIS
LIN {X -0.031,Y -392.864,Z 1294.187,A 0.000,B 0.000,C 90.000,E1 249.625} C_DIS
LIN {X 0.084,Y -402.028,Z 1294.169,A 0.000,B 0.000,C 90.000,E1 246.433} C_DIS
LIN {X -0.084,Y -412.751,Z 1294.152,A 0.000,B 0.000,C 90.000,E1 243.332} C_DIS
LIN {X 0.096,Y -424.381,Z 1294.136,A 0.000,B 0.000,C 90.000,E1 240.411} C_DIS
LIN {X 0.015,Y -437.565,Z 1294.120,A 0.000,B 0.000,C 90.000,E1 237.582} C_DIS
LIN {X -0.094,Y -452.395,Z 1294.104,A 0.000,B 0.000,C 90.000,E1 234.815} C_DIS
LIN {X -0.001,Y -453.304,Z 1294.104,A 0.000,B 0.000,C 90.000,E1 234.642} C_DIS
LIN {X -0.022,Y -454.464,Z 1294.102,A 0.000,B 0.000,C 90.000,E1 234.322} C_DIS
LIN {X 0.064,Y -455.169,Z 1294.100,A 0.000,B 0.000,C 90.000,E1 233.989} C_DIS
LIN {X -0.214,Y -455.656,Z 1294.098,A 0.000,B 0.000,C 90.000,E1 233.703} C_DIS
LIN {X -0.124,Y -456.232,Z 1294.095,A 0.000,B 0.000,C 90.000,E1 233.050} C_DIS
LIN {X 0.063,Y -456.610,Z 1294.089,A 0.000,B 0.000,C 90.000,E1 232.065} C_DIS
LIN {X 0.175,Y -456.552,Z 1294.084,A 0.000,B 0.000,C 90.000,E1 231.090} C_DIS
LIN {X -0.257,Y -455.968,Z 1294.075,A 0.000,B 0.000,C 90.000,E1 229.542} C_DIS
LIN {X -0.081,Y -455.402,Z 1294.064,A 0.000,B 0.000,C 90.000,E1 227.595} C_DIS
LIN {X 0.108,Y -454.896,Z 1294.052,A 0.000,B 0.000,C 90.000,E1 225.324} C_DIS
LIN {X -0.066,Y -454.812,Z 1294.041,A 0.000,B 0.000,C 90.000,E1 223.419} C_DIS
LIN {X 0.051,Y -456.238,Z 1294.014,A 0.000,B 0.000,C 90.000,E1 218.588} C_DIS
LIN {X -0.200,Y -457.576,Z 1294.002,A 0.000,B 0.000,C 90.000,E1 216.377} C_DIS
LIN {X 0.058,Y -460.641,Z 1293.983,A 0.000,B 0.000,C 90.000,E1 212.832} C_DIS
LIN {X 0.076,Y -463.471,Z 1293.968,A 0.000,B 0.000,C 90.000,E1 210.285} C_DIS
LIN {X -0.202,Y -466.265,Z 1293.956,A 0.000,B 0.000,C 90.000,E1 208.103} C_DIS
LIN {X 0.133,Y -469.667,Z 1293.942,A 0.000,B 0.000,C 90.000,E1 205.540} C_DIS
LIN {X -0.139,Y -471.974,Z 1293.933,A 0.000,B 0.000,C 90.000,E1 204.003} C_DIS
LIN {X 0.234,Y -475.158,Z 1293.921,A 0.000,B 0.000,C 90.000,E1 201.770} C_DIS
LIN {X -0.055,Y -477.533,Z 1293.912,A 0.000,B 0.000,C 90.000,E1 200.248} C_DIS
LIN {X -0.126,Y -479.529,Z 1293.906,A 0.000,B 0.000,C 90.000,E1 199.014} C_DIS
LIN {X -0.034,Y -482.051,Z 1293.897,A 0.000,B 0.000,C 90.000,E1 197.457} C_DIS
LIN {X 0.110,Y -484.611,Z 1293.888,A 0.000,B 0.000,C 90.000,E1 195.898} C_DIS
LIN {X 0.170,Y -487.127,Z 1293.880,A 0.000,B 0.000,C 90.000,E1 194.356} C_DIS
LIN {X 0.161,Y -489.678,Z 1293.871,A 0.000,B 0.000,C 90.000,E1 192.827} C_DIS
LIN {X -0.277,Y -491.663,Z 1293.865,A 0.000,B 0.000,C 90.000,E1 191.658} C_DIS
LIN {X 0.094,Y -494.676,Z 1293.854,A 0.000,B 0.000,C 90.000,E1 189.792} C_DIS
LIN {X 0.119,Y -497.191,Z 1293.846,A 0.000,B 0.000,C 90.000,E1 188.276} C_DIS
LIN {X 0.129,Y -499.151,Z 1293.839,A 0.000,B 0.000,C 90.000,E1 187.068} C_DIS
LIN {X 0.098,Y -501.614,Z 1293.831,A 0.000,B 0.000,C 90.000,E1 185.568} C_DIS
LIN {X 0.064,Y -503.862,Z 1293.823,A 0.000,B 0.000,C 90.000,E1 184.073} C_DIS
LIN {X 0.176,Y -505.684,Z 1293.816,A 0.000,B 0.000,C 90.000,E1 182.865} C_DIS
LIN {X 0.181,Y -507.785,Z 1293.808,A 0.000,B 0.000,C 90.000,E1 181.375} C_DIS
LIN {X 0.214,Y -509.628,Z 1293.800,A 0.000,B 0.000,C 90.000,E1 179.885} C_DIS
LIN {X -0.143,Y -510.946,Z 1293.793,A 0.000,B 0.000,C 90.000,E1 178.740} C_DIS
LIN {X -0.042,Y -512.403,Z 1293.785,A 0.000,B 0.000,C 90.000,E1 177.249} C_DIS
LIN {X 0.116,Y -513.574,Z 1293.776,A 0.000,B 0.000,C 90.000,E1 175.755} C_DIS
LIN {X -0.179,Y -514.180,Z 1293.770,A 0.000,B 0.000,C 90.000,E1 174.609} C_DIS
LIN {X 0.145,Y -514.505,Z 1293.763,A 0.000,B 0.000,C 90.000,E1 173.394} C_DIS
LIN {X -0.094,Y -514.647,Z 1293.757,A 0.000,B 0.000,C 90.000,E1 172.243} C_DIS
LIN {X -0.144,Y -514.598,Z 1293.754,A 0.000,B 0.000,C 90.000,E1 171.659} C_DIS
LIN {X 0.194,Y -514.077,Z 1293.747,A 0.000,B 0.000,C 90.000,E1 170.443} C_DIS
LIN {X 0.034,Y -513.632,Z 1293.742,A 0.000,B 0.000,C 90.000,E1 169.577} C_DIS
LIN {X -0.043,Y -512.864,Z 1293.737,A 0.000,B 0.000,C 90.000,E1 168.701} C_DIS
LIN {X -0.050,Y -511.535,Z 1293.731,A 0.000,B 0.000,C 90.000,E1 167.521} C_DIS
LIN {X -0.112,Y -510.683,Z 1293.727,A 0.000,B 0.000,C 90.000,E1 166.937} C_DIS
LIN {X -0.186,Y -508.283,Z 1293.719,A 0.000,B 0.000,C 90.000,E1 165.463} C_DIS
LIN {X -0.177,Y -505.377,Z 1293.711,A 0.000,B 0.000,C 90.000,E1 163.976} C_DIS
LIN {X -0.226,Y -502.243,Z 1293.703,A 0.000,B 0.000,C 90.000,E1 162.489} C_DIS
LIN {X -0.008,Y -496.889,Z 1293.689,A 0.000,B 0.000,C 90.000,E1 160.061} C_DIS
LIN {X 0.038,Y -494.365,Z 1293.683,A 0.000,B 0.000,C 90.000,E1 158.847} C_DIS
LIN {X -0.235,Y -492.277,Z 1293.676,A 0.000,B 0.000,C 90.000,E1 157.667} C_DIS
LIN {X -0.194,Y -491.967,Z 1293.674,A 0.000,B 0.000,C 90.000,E1 157.358} C_DIS
LIN {X -0.117,Y -492.436,Z 1293.671,A 0.000,B 0.000,C 90.000,E1 156.741} C_DIS
LIN {X 0.156,Y -493.350,Z 1293.667,A 0.000,B 0.000,C 90.000,E1 156.102} C_DIS
LIN {X -0.114,Y -495.418,Z 1293.664,A 0.000,B 0.000,C 90.000,E1 155.537} C_DIS
LIN {X -0.005,Y -496.865,Z 1293.663,A 0.000,B 0.000,C 90.000,E1 155.357} C_DIS
LIN {X -0.203,Y -497.824,Z 1293.662,A 0.000,B 0.000,C 90.000,E1 155.229} C_DIS
LIN {X -0.147,Y -499.053,Z 1293.661,A 0.000,B 0.000,C 90.000,E1 154.921} C_DIS
LIN {X 0.022,Y -501.654,Z 1293.659,A 0.000,B 0.000,C 90.000,E1 154.588} C_DIS
LIN {X 0.095,Y -508.341,Z 1293.655,A 0.000,B 0.000,C 90.000,E1 153.845} C_DIS
LIN {X -0.272,Y -515.820,Z 1293.650,A 0.000,B 0.000,C 90.000,E1 152.999} C_DIS
LIN {X 0.209,Y -520.305,Z 1293.647,A 0.000,B 0.000,C 90.000,E1 152.359} C_DIS
LIN {X -0.042,Y -523.537,Z 1293.644,A 0.000,B 0.000,C 90.000,E1 151.948} C_DIS
LIN {X -0.217,Y -527.371,Z 1293.641,A 0.000,B 0.000,C 90.000,E1 151.385} C_DIS
LIN {X -0.266,Y -531.496,Z 1293.637,A 0.000,B 0.000,C 90.000,E1 150.667} C_DIS
LIN {X 0.308,Y -532.157,Z 1293.636,A 0.000,B 0.000,C 90.000,E1 150.461} C_DIS
LIN {X -0.014,Y -535.583,Z 1293.633,A 0.000,B 0.000,C 90.000,E1 149.921} C_DIS
LIN {X -0.157,Y -536.693,Z 1293.632,A 0.000,B 0.000,C 90.000,E1 149.793} C_DIS
LIN {X 0.051,Y -539.263,Z 1293.631,A 0.000,B 0.000,C 90.000,E1 149.488} C_DIS
LIN {X 0.249,Y -543.733,Z 1293.628,A 0.000,B 0.000,C 90.000,E1 149.076} C_DIS
LIN {X 0.270,Y -550.974,Z 1293.625,A 0.000,B 0.000,C 90.000,E1 148.535} C_DIS
LIN {X 0.327,Y -558.496,Z 1293.622,A 0.000,B 0.000,C 90.000,E1 147.995} C_DIS
LIN {X 0.015,Y -564.355,Z 1293.620,A 0.000,B 0.000,C 90.000,E1 147.582} C_DIS
LIN {X 0.174,Y -574.194,Z 1293.616,A 0.000,B 0.000,C 90.000,E1 146.786} C_DIS
LIN {X 0.061,Y -579.937,Z 1293.613,A 0.000,B 0.000,C 90.000,E1 146.342} C_DIS
LIN {X -0.003,Y -585.376,Z 1293.610,A 0.000,B 0.000,C 90.000,E1 145.881} C_DIS
LIN {X 0.173,Y -592.116,Z 1293.607,A 0.000,B 0.000,C 90.000,E1 145.261} C_DIS
LIN {X 0.113,Y -597.088,Z 1293.604,A 0.000,B 0.000,C 90.000,E1 144.769} C_DIS
LIN {X -0.108,Y -600.732,Z 1293.602,A 0.000,B 0.000,C 90.000,E1 144.402} C_DIS
LIN {X 0.057,Y -605.308,Z 1293.599,A 0.000,B 0.000,C 90.000,E1 143.863} C_DIS
LIN {X 0.279,Y -609.339,Z 1293.597,A 0.000,B 0.000,C 90.000,E1 143.336} C_DIS
LIN {X 0.021,Y -614.833,Z 1293.592,A 0.000,B 0.000,C 90.000,E1 142.603} C_DIS
LIN {X -0.238,Y -618.289,Z 1293.589,A 0.000,B 0.000,C 90.000,E1 142.110} C_DIS
LIN {X -0.127,Y -622.282,Z 1293.586,A 0.000,B 0.000,C 90.000,E1 141.457} C_DIS
LIN {X -0.315,Y -624.592,Z 1293.584,A 0.000,B 0.000,C 90.000,E1 141.090} C_DIS
LIN {X -0.153,Y -628.193,Z 1293.580,A 0.000,B 0.000,C 90.000,E1 140.436} C_DIS
LIN {X 0.069,Y -632.692,Z 1293.575,A 0.000,B 0.000,C 90.000,E1 139.542} C_DIS
LIN {X -0.295,Y -636.916,Z 1293.570,A 0.000,B 0.000,C 90.000,E1 138.690} C_DIS
LIN {X -0.115,Y -640.259,Z 1293.566,A 0.000,B 0.000,C 90.000,E1 137.919} C_DIS
LIN {X 0.021,Y -644.501,Z 1293.561,A 0.000,B 0.000,C 90.000,E1 136.905} C_DIS
LIN {X 0.152,Y -649.533,Z 1293.554,A 0.000,B 0.000,C 90.000,E1 135.648} C_DIS
LIN {X -0.102,Y -654.487,Z 1293.547,A 0.000,B 0.000,C 90.000,E1 134.433} C_DIS
LIN {X 0.170,Y -660.272,Z 1293.539,A 0.000,B 0.000,C 90.000,E1 132.933} C_DIS
LIN {X 0.084,Y -664.101,Z 1293.533,A 0.000,B 0.000,C 90.000,E1 131.962} C_DIS
LIN {X 0.088,Y -668.696,Z 1293.526,A 0.000,B 0.000,C 90.000,E1 130.744} C_DIS
LIN {X 0.157,Y -671.326,Z 1293.522,A 0.000,B 0.000,C 90.000,E1 130.011} C_DIS
LIN {X -0.151,Y -675.423,Z 1293.516,A 0.000,B 0.000,C 90.000,E1 128.830} C_DIS
LIN {X 0.138,Y -679.275,Z 1293.509,A 0.000,B 0.000,C 90.000,E1 127.604} C_DIS
LIN {X -0.056,Y -682.783,Z 1293.502,A 0.000,B 0.000,C 90.000,E1 126.423} C_DIS
LIN {X -0.058,Y -685.922,Z 1293.496,A 0.000,B 0.000,C 90.000,E1 125.231} C_DIS
LIN {X -0.029,Y -688.257,Z 1293.490,A 0.000,B 0.000,C 90.000,E1 124.278} C_DIS
LIN {X 0.420,Y -690.316,Z 1293.485,A 0.000,B 0.000,C 90.000,E1 123.293} C_DIS
LIN {X -0.445,Y -692.071,Z 1293.480,A 0.000,B 0.000,C 90.000,E1 122.418} C_DIS
LIN {X -0.331,Y -693.673,Z 1293.475,A 0.000,B 0.000,C 90.000,E1 121.465} C_DIS
LIN {X 0.286,Y -695.871,Z 1293.467,A 0.000,B 0.000,C 90.000,E1 120.001} C_DIS
LIN {X 0.088,Y -697.155,Z 1293.462,A 0.000,B 0.000,C 90.000,E1 119.077} C_DIS
LIN {X 0.253,Y -697.990,Z 1293.458,A 0.000,B 0.000,C 90.000,E1 118.359} C_DIS
LIN {X 0.426,Y -698.586,Z 1293.454,A 0.000,B 0.000,C 90.000,E1 117.641} C_DIS
LIN {X -0.338,Y -698.967,Z 1293.450,A 0.000,B 0.000,C 90.000,E1 117.001} C_DIS
LIN {X 0.104,Y -699.109,Z 1293.445,A 0.000,B 0.000,C 90.000,E1 116.027} C_DIS
LIN {X -0.029,Y -698.808,Z 1293.441,A 0.000,B 0.000,C 90.000,E1 115.335} C_DIS
LIN {X 0.209,Y -698.428,Z 1293.438,A 0.000,B 0.000,C 90.000,E1 114.847} C_DIS
LIN {X 0.103,Y -697.651,Z 1293.436,A 0.000,B 0.000,C 90.000,E1 114.387} C_DIS
LIN {X 0.078,Y -697.140,Z 1293.434,A 0.000,B 0.000,C 90.000,E1 114.155} C_DIS
LIN {X -0.042,Y -695.484,Z 1293.432,A 0.000,B 0.000,C 90.000,E1 113.695} C_DIS
LIN {X 0.085,Y -694.957,Z 1293.431,A 0.000,B 0.000,C 90.000,E1 113.567} C_DIS
LIN {X 0.303,Y -691.723,Z 1293.428,A 0.000,B 0.000,C 90.000,E1 113.078} C_DIS
LIN {X 0.423,Y -690.802,Z 1293.428,A 0.000,B 0.000,C 90.000,E1 112.950} C_DIS
LIN {X -0.363,Y -689.429,Z 1293.427,A 0.000,B 0.000,C 90.000,E1 112.898} C_DIS
LIN {X 0.139,Y -683.194,Z 1293.425,A 0.000,B 0.000,C 90.000,E1 112.461} C_DIS
LIN {X -0.102,Y -681.130,Z 1293.424,A 0.000,B 0.000,C 90.000,E1 112.386} C_DIS
LIN {X -0.358,Y -678.501,Z 1293.424,A 0.000,B 0.000,C 90.000,E1 112.333} C_DIS
LIN {X 0.272,Y -675.268,Z 1293.424,A 0.000,B 0.000,C 90.000,E1 112.206} C_DIS
LIN {X -0.187,Y -671.757,Z 1293.423,A 0.000,B 0.000,C 90.000,E1 112.153} C_DIS
LIN {X 0.138,Y -670.200,Z 1293.423,A 0.000,B 0.000,C 90.000,E1 112.099} C_DIS
LIN {X 0.286,Y -663.377,Z 1293.423,A 0.000,B 0.000,C 90.000,E1 112.025} C_DIS
LIN {X 0.218,Y -648.593,Z 1293.422,A 0.000,B 0.000,C 90.000,E1 112.025} C_DIS
LIN {X -0.170,Y -643.460,Z 1293.422,A 0.000,B 0.000,C 90.000,E1 112.025} C_DIS
LIN {X 0.103,Y -639.413,Z 1293.422,A 0.000,B 0.000,C 90.000,E1 111.897} C_DIS
LIN {X 0.049,Y -639.324,Z 1293.422,A 0.000,B 0.000,C 90.000,E1 111.897} C_DIS
LIN {X -0.013,Y -640.834,Z 1293.420,A 0.000,B 0.000,C 90.000,E1 111.589} C_DIS
LIN {X -0.023,Y -641.924,Z 1293.419,A 0.000,B 0.000,C 90.000,E1 111.408} C_DIS
LIN {X -0.240,Y -649.464,Z 1293.413,A 0.000,B 0.000,C 90.000,E1 110.429} C_DIS
LIN {X -0.167,Y -651.186,Z 1293.412,A 0.000,B 0.000,C 90.000,E1 110.174} C_DIS
LIN {X 0.211,Y -655.138,Z 1293.409,A 0.000,B 0.000,C 90.000,E1 109.523} C_DIS
LIN {X 0.111,Y -659.780,Z 1293.404,A 0.000,B 0.000,C 90.000,E1 108.671} C_DIS
LIN {X -0.001,Y -663.226,Z 1293.400,A 0.000,B 0.000,C 90.000,E1 107.946} C_DIS
LIN {X -0.082,Y -666.227,Z 1293.396,A 0.000,B 0.000,C 90.000,E1 107.221} C_DIS
LIN {X -0.059,Y -668.067,Z 1293.393,A 0.000,B 0.000,C 90.000,E1 106.732} C_DIS
LIN {X -0.290,Y -670.374,Z 1293.389,A 0.000,B 0.000,C 90.000,E1 106.024} C_DIS
LIN {X 0.332,Y -672.249,Z 1293.385,A 0.000,B 0.000,C 90.000,E1 105.245} C_DIS
LIN {X 0.148,Y -673.844,Z 1293.381,A 0.000,B 0.000,C 90.000,E1 104.537} C_DIS
LIN {X 0.034,Y -674.679,Z 1293.378,A 0.000,B 0.000,C 90.000,E1 104.064} C_DIS
LIN {X -0.127,Y -675.697,Z 1293.374,A 0.000,B 0.000,C 90.000,E1 103.355} C_DIS
LIN {X -0.281,Y -676.322,Z 1293.370,A 0.000,B 0.000,C 90.000,E1 102.647} C_DIS
LIN {X 0.228,Y -676.507,Z 1293.366,A 0.000,B 0.000,C 90.000,E1 101.883} C_DIS
LIN {X -0.010,Y -676.439,Z 1293.364,A 0.000,B 0.000,C 90.000,E1 101.422} C_DIS
LIN {X -0.112,Y -676.197,Z 1293.361,A 0.000,B 0.000,C 90.000,E1 100.950} C_DIS
LIN {X -0.344,Y -675.748,Z 1293.358,A 0.000,B 0.000,C 90.000,E1 100.489} C_DIS
LIN {X 0.210,Y -675.106,Z 1293.355,A 0.000,B 0.000,C 90.000,E1 99.962} C_DIS
LIN {X -0.022,Y -674.143,Z 1293.353,A 0.000,B 0.000,C 90.000,E1 99.500} C_DIS
LIN {X -0.085,Y -673.598,Z 1293.351,A 0.000,B 0.000,C 90.000,E1 99.265} C_DIS
LIN {X -0.323,Y -672.221,Z 1293.349,A 0.000,B 0.000,C 90.000,E1 98.803} C_DIS
LIN {X 0.196,Y -670.539,Z 1293.346,A 0.000,B 0.000,C 90.000,E1 98.276} C_DIS
LIN {X -0.060,Y -668.500,Z 1293.343,A 0.000,B 0.000,C 90.000,E1 97.814} C_DIS
LIN {X 0.335,Y -666.164,Z 1293.341,A 0.000,B 0.000,C 90.000,E1 97.296} C_DIS
LIN {X 0.146,Y -664.233,Z 1293.339,A 0.000,B 0.000,C 90.000,E1 96.947} C_DIS
LIN {X -0.150,Y -661.416,Z 1293.336,A 0.000,B 0.000,C 90.000,E1 96.486} C_DIS
LIN {X 0.193,Y -658.376,Z 1293.333,A 0.000,B 0.000,C 90.000,E1 95.967} C_DIS
LIN {X -0.243,Y -654.021,Z 1293.330,A 0.000,B 0.000,C 90.000,E1 95.391} C_DIS
LIN {X -0.010,Y -650.239,Z 1293.327,A 0.000,B 0.000,C 90.000,E1 94.878} C_DIS
LIN {X 0.254,Y -646.155,Z 1293.324,A 0.000,B 0.000,C 90.000,E1 94.359} C_DIS
LIN {X -0.275,Y -640.430,Z 1293.321,A 0.000,B 0.000,C 90.000,E1 93.784} C_DIS
LIN {X -0.238,Y -633.158,Z 1293.317,A 0.000,B 0.000,C 90.000,E1 93.037} C_DIS
LIN {X -0.268,Y -624.491,Z 1293.312,A 0.000,B 0.000,C 90.000,E1 92.178} C_DIS
LIN {X 0.122,Y -619.170,Z 1293.309,A 0.000,B 0.000,C 90.000,E1 91.661} C_DIS
LIN {X 0.040,Y -616.379,Z 1293.308,A 0.000,B 0.000,C 90.000,E1 91.432} C_DIS
LIN {X -0.146,Y -609.005,Z 1293.305,A 0.000,B 0.000,C 90.000,E1 90.917} C_DIS
LIN {X -0.027,Y -602.882,Z 1293.303,A 0.000,B 0.000,C 90.000,E1 90.516} C_DIS
LIN {X 0.274,Y -596.352,Z 1293.301,A 0.000,B 0.000,C 90.000,E1 90.115} C_DIS
LIN {X -0.216,Y -589.420,Z 1293.299,A 0.000,B 0.000,C 90.000,E1 89.828} C_DIS
LIN {X -0.227,Y -582.122,Z 1293.297,A 0.000,B 0.000,C 90.000,E1 89.542} C_DIS
LIN {X 0.203,Y -576.703,Z 1293.296,A 0.000,B 0.000,C 90.000,E1 89.312} C_DIS
LIN {X 0.135,Y -572.954,Z 1293.295,A 0.000,B 0.000,C 90.000,E1 89.141} C_DIS
LIN {X 0.107,Y -571.848,Z 1293.295,A 0.000,B 0.000,C 90.000,E1 89.083} C_DIS
LIN {X -0.280,Y -570.163,Z 1293.294,A 0.000,B 0.000,C 90.000,E1 88.969} C_DIS
LIN {X 0.252,Y -570.139,Z 1293.294,A 0.000,B 0.000,C 90.000,E1 88.912} C_DIS
LIN {X -0.102,Y -569.750,Z 1293.293,A 0.000,B 0.000,C 90.000,E1 88.797} C_DIS
LIN {X -0.227,Y -569.638,Z 1293.292,A 0.000,B 0.000,C 90.000,E1 88.568} C_DIS
LIN {X -0.100,Y -569.631,Z 1293.290,A 0.000,B 0.000,C 90.000,E1 88.282} C_DIS
LIN {X 0.251,Y -572.119,Z 1293.274,A 0.000,B 0.000,C 90.000,E1 85.241} C_DIS
LIN {X -0.222,Y -574.517,Z 1293.262,A 0.000,B 0.000,C 90.000,E1 83.109} C_DIS
LIN {X -0.109,Y -576.788,Z 1293.251,A 0.000,B 0.000,C 90.000,E1 81.197} C_DIS
LIN {X 0.293,Y -578.387,Z 1293.244,A 0.000,B 0.000,C 90.000,E1 79.803} C_DIS
LIN {X 0.149,Y -579.768,Z 1293.236,A 0.000,B 0.000,C 90.000,E1 78.465} C_DIS
LIN {X 0.140,Y -581.000,Z 1293.229,A 0.000,B 0.000,C 90.000,E1 77.117} C_DIS
LIN {X 0.287,Y -582.121,Z 1293.221,A 0.000,B 0.000,C 90.000,E1 75.755} C_DIS
LIN {X -0.104,Y -583.133,Z 1293.214,A 0.000,B 0.000,C 90.000,E1 74.448} C_DIS
LIN {X 0.140,Y -584.360,Z 1293.203,A 0.000,B 0.000,C 90.000,E1 72.543} C_DIS
LIN {X -0.054,Y -585.296,Z 1293.196,A 0.000,B 0.000,C 90.000,E1 71.221} C_DIS
LIN {X -0.101,Y -586.503,Z 1293.184,A 0.000,B 0.000,C 90.000,E1 69.082} C_DIS
LIN {X 0.102,Y -587.829,Z 1293.172,A 0.000,B 0.000,C 90.000,E1 66.922} C_DIS
LIN {X 0.135,Y -589.149,Z 1293.161,A 0.000,B 0.000,C 90.000,E1 65.049} C_DIS
LIN {X 0.015,Y -590.320,Z 1293.153,A 0.000,B 0.000,C 90.000,E1 63.461} C_DIS
LIN {X 0.261,Y -592.152,Z 1293.141,A 0.000,B 0.000,C 90.000,E1 61.307} C_DIS
LIN {X 0.150,Y -594.028,Z 1293.130,A 0.000,B 0.000,C 90.000,E1 59.459} C_DIS
LIN {X 0.169,Y -595.656,Z 1293.122,A 0.000,B 0.000,C 90.000,E1 57.867} C_DIS
LIN {X 0.026,Y -597.306,Z 1293.113,A 0.000,B 0.000,C 90.000,E1 56.294} C_DIS
LIN {X 0.017,Y -598.686,Z 1293.105,A 0.000,B 0.000,C 90.000,E1 54.975} C_DIS
LIN {X -0.216,Y -600.136,Z 1293.097,A 0.000,B 0.000,C 90.000,E1 53.417} C_DIS
LIN {X 0.168,Y -601.205,Z 1293.089,A 0.000,B 0.000,C 90.000,E1 52.065} C_DIS
LIN {X 0.218,Y -602.140,Z 1293.083,A 0.000,B 0.000,C 90.000,E1 51.009} C_DIS
LIN {X -0.095,Y -602.772,Z 1293.078,A 0.000,B 0.000,C 90.000,E1 49.989} C_DIS
LIN {X -0.222,Y -603.456,Z 1293.070,A 0.000,B 0.000,C 90.000,E1 48.690} C_DIS
LIN {X 0.066,Y -603.710,Z 1293.066,A 0.000,B 0.000,C 90.000,E1 47.877} C_DIS
LIN {X 0.158,Y -604.182,Z 1293.057,A 0.000,B 0.000,C 90.000,E1 46.296} C_DIS
LIN {X 0.223,Y -604.268,Z 1293.052,A 0.000,B 0.000,C 90.000,E1 45.243} C_DIS
LIN {X 0.290,Y -604.240,Z 1293.046,A 0.000,B 0.000,C 90.000,E1 44.190} C_DIS
LIN {X -0.062,Y -603.984,Z 1293.040,A 0.000,B 0.000,C 90.000,E1 43.176} C_DIS
LIN {X 0.236,Y -603.627,Z 1293.033,A 0.000,B 0.000,C 90.000,E1 41.838} C_DIS
LIN {X 0.077,Y -603.309,Z 1293.028,A 0.000,B 0.000,C 90.000,E1 41.067} C_DIS
LIN {X -0.017,Y -602.450,Z 1293.018,A 0.000,B 0.000,C 90.000,E1 39.241} C_DIS
LIN {X -0.112,Y -601.988,Z 1293.014,A 0.000,B 0.000,C 90.000,E1 38.463} C_DIS
LIN {X -0.179,Y -600.853,Z 1293.006,A 0.000,B 0.000,C 90.000,E1 37.156} C_DIS
LIN {X -0.031,Y -599.635,Z 1293.000,A 0.000,B 0.000,C 90.000,E1 36.091} C_DIS
LIN {X 0.098,Y -598.194,Z 1292.995,A 0.000,B 0.000,C 90.000,E1 35.025} C_DIS
LIN {X -0.136,Y -596.341,Z 1292.989,A 0.000,B 0.000,C 90.000,E1 33.992} C_DIS
LIN {X 0.106,Y -594.292,Z 1292.983,A 0.000,B 0.000,C 90.000,E1 32.911} C_DIS
LIN {X -0.282,Y -593.102,Z 1292.980,A 0.000,B 0.000,C 90.000,E1 32.418} C_DIS
LIN {X 0.024,Y -590.973,Z 1292.976,A 0.000,B 0.000,C 90.000,E1 31.592} C_DIS
LIN {X -0.117,Y -587.752,Z 1292.970,A 0.000,B 0.000,C 90.000,E1 30.541} C_DIS
LIN {X -0.173,Y -584.784,Z 1292.965,A 0.000,B 0.000,C 90.000,E1 29.745} C_DIS
LIN {X -0.133,Y -582.627,Z 1292.962,A 0.000,B 0.000,C 90.000,E1 29.205} C_DIS
LIN {X 0.191,Y -578.380,Z 1292.957,A 0.000,B 0.000,C 90.000,E1 28.231} C_DIS
LIN {X 0.020,Y -574.192,Z 1292.953,A 0.000,B 0.000,C 90.000,E1 27.436} C_DIS
LIN {X 0.213,Y -571.093,Z 1292.949,A 0.000,B 0.000,C 90.000,E1 26.873} C_DIS
LIN {X -0.120,Y -567.837,Z 1292.946,A 0.000,B 0.000,C 90.000,E1 26.360} C_DIS
LIN {X -0.148,Y -562.600,Z 1292.942,A 0.000,B 0.000,C 90.000,E1 25.540} C_DIS
LIN {X 0.004,Y -556.757,Z 1292.937,A 0.000,B 0.000,C 90.000,E1 24.695} C_DIS
LIN {X 0.079,Y -552.556,Z 1292.934,A 0.000,B 0.000,C 90.000,E1 24.131} C_DIS
LIN {X 0.122,Y -548.048,Z 1292.931,A 0.000,B 0.000,C 90.000,E1 23.567} C_DIS
LIN {X 0.036,Y -539.587,Z 1292.926,A 0.000,B 0.000,C 90.000,E1 22.589} C_DIS
LIN {X -0.011,Y -534.558,Z 1292.922,A 0.000,B 0.000,C 90.000,E1 22.025} C_DIS
LIN {X -0.001,Y -525.483,Z 1292.917,A 0.000,B 0.000,C 90.000,E1 21.046} C_DIS
LIN {X -0.095,Y -518.823,Z 1292.913,A 0.000,B 0.000,C 90.000,E1 20.355} C_DIS
LIN {X 0.192,Y -512.055,Z 1292.909,A 0.000,B 0.000,C 90.000,E1 19.631} C_DIS
LIN {X -0.182,Y -503.800,Z 1292.905,A 0.000,B 0.000,C 90.000,E1 18.852} C_DIS
LIN {X 0.005,Y -494.062,Z 1292.899,A 0.000,B 0.000,C 90.000,E1 17.873} C_DIS
LIN {X 0.282,Y -484.282,Z 1292.894,A 0.000,B 0.000,C 90.000,E1 16.913} C_DIS
LIN {X -0.070,Y -473.935,Z 1292.889,A 0.000,B 0.000,C 90.000,E1 16.024} C_DIS
LIN {X 0.218,Y -463.673,Z 1292.884,A 0.000,B 0.000,C 90.000,E1 15.064} C_DIS
LIN {X -0.119,Y -453.522,Z 1292.879,A 0.000,B 0.000,C 90.000,E1 14.175} C_DIS
LIN {X 0.008,Y -431.949,Z 1292.867,A 0.000,B 0.000,C 90.000,E1 12.063} C_DIS
LIN {X -0.107,Y -416.147,Z 1292.858,A 0.000,B 0.000,C 90.000,E1 10.423} C_DIS
LIN {X 0.106,Y -403.238,Z 1292.850,A 0.000,B 0.000,C 90.000,E1 8.973} C_DIS
LIN {X -0.036,Y -399.199,Z 1292.847,A 0.000,B 0.000,C 90.000,E1 8.511} C_DIS
LIN {X -0.005,Y -396.588,Z 1292.845,A 0.000,B 0.000,C 90.000,E1 8.163} C_DIS
LIN {X 0.129,Y -395.230,Z 1292.844,A 0.000,B 0.000,C 90.000,E1 7.871} C_DIS
LIN {X 0.090,Y -395.223,Z 1292.844,A 0.000,B 0.000,C 90.000,E1 7.871} C_DIS
LIN {X 0.053,Y -395.226,Z 1292.844,A 0.000,B 0.000,C 90.000,E1 7.871} C_DIS
LIN {X 0.050,Y -396.282,Z 1292.843,A 0.000,B 0.000,C 90.000,E1 7.701} C_DIS
LIN {X -0.160,Y -399.876,Z 1292.841,A 0.000,B 0.000,C 90.000,E1 7.409} C_DIS
LIN {X 0.083,Y -407.956,Z 1292.838,A 0.000,B 0.000,C 90.000,E1 6.891} C_DIS
LIN {X 0.014,Y -411.223,Z 1292.837,A 0.000,B 0.000,C 90.000,E1 6.720} C_DIS
LIN {X -0.004,Y -419.039,Z 1292.834,A 0.000,B 0.000,C 90.000,E1 6.201} C_DIS
LIN {X 0.082,Y -423.879,Z 1292.833,A 0.000,B 0.000,C 90.000,E1 5.853} C_DIS
LIN {X -0.066,Y -431.598,Z 1292.829,A 0.000,B 0.000,C 90.000,E1 5.277} C_DIS
LIN {X -0.015,Y -439.370,Z 1292.826,A 0.000,B 0.000,C 90.000,E1 4.645} C_DIS
LIN {X 0.170,Y -448.512,Z 1292.822,A 0.000,B 0.000,C 90.000,E1 3.841} C_DIS
LIN {X 0.014,Y -455.776,Z 1292.818,A 0.000,B 0.000,C 90.000,E1 3.212} C_DIS
LIN {X 0.226,Y -461.481,Z 1292.815,A 0.000,B 0.000,C 90.000,E1 2.636} C_DIS
LIN {X -0.184,Y -467.084,Z 1292.812,A 0.000,B 0.000,C 90.000,E1 2.121} C_DIS
LIN {X -0.007,Y -473.684,Z 1292.808,A 0.000,B 0.000,C 90.000,E1 1.375} C_DIS
LIN {X 0.113,Y -478.790,Z 1292.804,A 0.000,B 0.000,C 90.000,E1 0.745} C_DIS
LIN {X -0.228,Y -483.626,Z 1292.801,A 0.000,B 0.000,C 90.000,E1 0.172} C_DIS
LIN {X 0.169,Y -489.505,Z 1292.796,A 0.000,B 0.000,C 90.000,E1 359.312} C_DIS
LIN {X 0.016,Y -494.554,Z 1292.792,A 0.000,B 0.000,C 90.000,E1 358.568} C_DIS
LIN {X 0.241,Y -498.400,Z 1292.789,A 0.000,B 0.000,C 90.000,E1 357.936} C_DIS
LIN {X -0.144,Y -503.617,Z 1292.784,A 0.000,B 0.000,C 90.000,E1 357.078} C_DIS
LIN {X 0.159,Y -506.969,Z 1292.780,A 0.000,B 0.000,C 90.000,E1 356.445} C_DIS
LIN {X 0.192,Y -510.840,Z 1292.776,A 0.000,B 0.000,C 90.000,E1 355.698} C_DIS
LIN {X -0.040,Y -515.189,Z 1292.771,A 0.000,B 0.000,C 90.000,E1 354.837} C_DIS
LIN {X 0.142,Y -517.263,Z 1292.769,A 0.000,B 0.000,C 90.000,E1 354.375} C_DIS
LIN {X -0.028,Y -521.045,Z 1292.764,A 0.000,B 0.000,C 90.000,E1 353.514} C_DIS
LIN {X -0.039,Y -523.426,Z 1292.761,A 0.000,B 0.000,C 90.000,E1 352.932} C_DIS
LIN {X -0.099,Y -525.640,Z 1292.758,A 0.000,B 0.000,C 90.000,E1 352.356} C_DIS
LIN {X -0.127,Y -528.708,Z 1292.753,A 0.000,B 0.000,C 90.000,E1 351.489} C_DIS
LIN {X -0.125,Y -531.524,Z 1292.748,A 0.000,B 0.000,C 90.000,E1 350.622} C_DIS
LIN {X -0.005,Y -534.097,Z 1292.743,A 0.000,B 0.000,C 90.000,E1 349.746} C_DIS
LIN {X 0.148,Y -536.396,Z 1292.738,A 0.000,B 0.000,C 90.000,E1 348.870} C_DIS
LIN {X -0.132,Y -539.157,Z 1292.732,A 0.000,B 0.000,C 90.000,E1 347.757} C_DIS
LIN {X 0.076,Y -540.973,Z 1292.727,A 0.000,B 0.000,C 90.000,E1 346.881} C_DIS
LIN {X -0.098,Y -542.573,Z 1292.723,A 0.000,B 0.000,C 90.000,E1 346.047} C_DIS
LIN {X 0.138,Y -543.923,Z 1292.718,A 0.000,B 0.000,C 90.000,E1 345.172} C_DIS
LIN {X 0.080,Y -545.392,Z 1292.711,A 0.000,B 0.000,C 90.000,E1 344.047} C_DIS
LIN {X 0.192,Y -546.396,Z 1292.705,A 0.000,B 0.000,C 90.000,E1 342.906} C_DIS
LIN {X 0.243,Y -546.915,Z 1292.700,A 0.000,B 0.000,C 90.000,E1 342.054} C_DIS
LIN {X 0.130,Y -547.181,Z 1292.696,A 0.000,B 0.000,C 90.000,E1 341.221} C_DIS
LIN {X 0.192,Y -547.072,Z 1292.691,A 0.000,B 0.000,C 90.000,E1 340.369} C_DIS
LIN {X -0.259,Y -546.710,Z 1292.686,A 0.000,B 0.000,C 90.000,E1 339.571} C_DIS
LIN {X -0.202,Y -545.978,Z 1292.682,A 0.000,B 0.000,C 90.000,E1 338.720} C_DIS
LIN {X -0.205,Y -545.343,Z 1292.679,A 0.000,B 0.000,C 90.000,E1 338.156} C_DIS
LIN {X 0.073,Y -543.638,Z 1292.672,A 0.000,B 0.000,C 90.000,E1 336.997} C_DIS
LIN {X -0.204,Y -542.316,Z 1292.668,A 0.000,B 0.000,C 90.000,E1 336.177} C_DIS
LIN {X -0.229,Y -540.727,Z 1292.664,A 0.000,B 0.000,C 90.000,E1 335.613} C_DIS
LIN {X 0.000,Y -540.156,Z 1292.663,A 0.000,B 0.000,C 90.000,E1 335.305} C_DIS
LIN {X -0.081,Y -537.734,Z 1292.658,A 0.000,B 0.000,C 90.000,E1 334.460} C_DIS
LIN {X 0.224,Y -533.213,Z 1292.650,A 0.000,B 0.000,C 90.000,E1 332.999} C_DIS
LIN {X -0.208,Y -529.465,Z 1292.644,A 0.000,B 0.000,C 90.000,E1 331.897} C_DIS
LIN {X 0.073,Y -526.193,Z 1292.639,A 0.000,B 0.000,C 90.000,E1 331.001} C_DIS
LIN {X 0.109,Y -522.298,Z 1292.634,A 0.000,B 0.000,C 90.000,E1 330.127} C_DIS
LIN {X -0.159,Y -518.048,Z 1292.629,A 0.000,B 0.000,C 90.000,E1 329.282} C_DIS
LIN {X -0.036,Y -514.275,Z 1292.625,A 0.000,B 0.000,C 90.000,E1 328.535} C_DIS
LIN {X -0.079,Y -506.058,Z 1292.616,A 0.000,B 0.000,C 90.000,E1 326.914} C_DIS
LIN {X 0.130,Y -503.417,Z 1292.613,A 0.000,B 0.000,C 90.000,E1 326.294} C_DIS
LIN {X -0.097,Y -501.196,Z 1292.609,A 0.000,B 0.000,C 90.000,E1 325.722} C_DIS
LIN {X -0.042,Y -498.704,Z 1292.605,A 0.000,B 0.000,C 90.000,E1 324.815} C_DIS
LIN {X -0.018,Y -497.091,Z 1292.599,A 0.000,B 0.000,C 90.000,E1 323.909} C_DIS
LIN {X 0.144,Y -495.869,Z 1292.593,A 0.000,B 0.000,C 90.000,E1 322.683} C_DIS
LIN {X 0.123,Y -495.308,Z 1292.588,A 0.000,B 0.000,C 90.000,E1 321.778} C_DIS
LIN {X 0.170,Y -495.315,Z 1292.566,A 0.000,B 0.000,C 90.000,E1 317.838} C_DIS
LIN {X -0.096,Y -495.514,Z 1292.556,A 0.000,B 0.000,C 90.000,E1 316.053} C_DIS
LIN {X 0.139,Y -495.695,Z 1292.547,A 0.000,B 0.000,C 90.000,E1 314.514} C_DIS
LIN {X 0.185,Y -495.771,Z 1292.541,A 0.000,B 0.000,C 90.000,E1 313.299} C_DIS
LIN {X 0.070,Y -495.513,Z 1292.536,A 0.000,B 0.000,C 90.000,E1 312.405} C_DIS
LIN {X -0.262,Y -495.052,Z 1292.532,A 0.000,B 0.000,C 90.000,E1 311.838} C_DIS
LIN {X -0.229,Y -494.304,Z 1292.529,A 0.000,B 0.000,C 90.000,E1 311.229} C_DIS
LIN {X -0.052,Y -493.730,Z 1292.527,A 0.000,B 0.000,C 90.000,E1 310.906} C_DIS
LIN {X -0.200,Y -492.978,Z 1292.526,A 0.000,B 0.000,C 90.000,E1 310.620} C_DIS
LIN {X -0.031,Y -491.881,Z 1292.524,A 0.000,B 0.000,C 90.000,E1 310.297} C_DIS
LIN {X -0.264,Y -491.020,Z 1292.523,A 0.000,B 0.000,C 90.000,E1 310.172} C_DIS
LIN {X 0.031,Y -473.023,Z 1292.509,A 0.000,B 0.000,C 90.000,E1 307.523} C_DIS
LIN {X 0.210,Y -456.832,Z 1292.494,A 0.000,B 0.000,C 90.000,E1 304.818} C_DIS
LIN {X 0.113,Y -442.343,Z 1292.478,A 0.000,B 0.000,C 90.000,E1 302.084} C_DIS
LIN {X 0.082,Y -429.452,Z 1292.463,A 0.000,B 0.000,C 90.000,E1 299.283} C_DIS
LIN {X -0.142,Y -417.451,Z 1292.446,A 0.000,B 0.000,C 90.000,E1 296.283} C_DIS
LIN {X -0.126,Y -406.527,Z 1292.428,A 0.000,B 0.000,C 90.000,E1 293.025} C_DIS
LIN {X -0.033,Y -401.979,Z 1292.419,A 0.000,B 0.000,C 90.000,E1 291.461} C_DIS
LIN {X -0.070,Y -401.970,Z 1292.419,A 0.000,B 0.000,C 90.000,E1 291.461} C_DIS
LIN {X -0.058,Y -404.695,Z 1292.395,A 0.000,B 0.000,C 90.000,E1 287.094} C_DIS
LIN {X -0.164,Y -404.779,Z 1292.385,A 0.000,B 0.000,C 90.000,E1 285.371} C_DIS
LIN {X -0.066,Y -406.123,Z 1292.364,A 0.000,B 0.000,C 90.000,E1 281.535} C_DIS
LIN {X -0.034,Y -405.828,Z 1292.358,A 0.000,B 0.000,C 90.000,E1 280.489} C_DIS
LIN {X 0.027,Y -405.688,Z 1292.333,A 0.000,B 0.000,C 90.000,E1 275.967} C_DIS
LIN {X 0.065,Y -403.472,Z 1292.304,A 0.000,B 0.000,C 90.000,E1 270.745} C_DIS
LIN {X 0.032,Y -403.260,Z 1292.302,A 0.000,B 0.000,C 90.000,E1 270.401} C_DIS
LIN {X -0.186,Y -398.885,Z 1292.271,A 0.000,B 0.000,C 90.000,E1 264.837} C_DIS
LIN {X 0.109,Y -393.355,Z 1292.244,A 0.000,B 0.000,C 90.000,E1 259.859} C_DIS
LIN {X 0.030,Y -392.789,Z 1292.240,A 0.000,B 0.000,C 90.000,E1 259.162} C_DIS
LIN {X -0.103,Y -387.173,Z 1292.218,A 0.000,B 0.000,C 90.000,E1 255.283} C_DIS
LIN {X -0.141,Y -387.169,Z 1292.218,A 0.000,B 0.000,C 90.000,E1 255.283} C_DIS
LIN {X -0.043,Y -394.655,Z 1292.198,A 0.000,B 0.000,C 90.000,E1 251.692} C_DIS
LIN {X 0.088,Y -403.896,Z 1292.179,A 0.000,B 0.000,C 90.000,E1 248.156} C_DIS
LIN {X 0.254,Y -414.402,Z 1292.161,A 0.000,B 0.000,C 90.000,E1 244.845} C_DIS
LIN {X 0.010,Y -425.980,Z 1292.144,A 0.000,B 0.000,C 90.000,E1 241.820} C_DIS
LIN {X -0.082,Y -438.455,Z 1292.128,A 0.000,B 0.000,C 90.000,E1 238.997} C_DIS
LIN {X -0.045,Y -452.517,Z 1292.112,A 0.000,B 0.000,C 90.000,E1 236.215} C_DIS
LIN {X 0.040,Y -454.279,Z 1292.110,A 0.000,B 0.000,C 90.000,E1 235.881} C_DIS
LIN {X 0.024,Y -455.022,Z 1292.110,A 0.000,B 0.000,C 90.000,E1 235.722} C_DIS
LIN {X 0.121,Y -455.937,Z 1292.108,A 0.000,B 0.000,C 90.000,E1 235.388} C_DIS
LIN {X -0.157,Y -456.519,Z 1292.106,A 0.000,B 0.000,C 90.000,E1 235.102} C_DIS
LIN {X 0.043,Y -457.219,Z 1292.103,A 0.000,B 0.000,C 90.000,E1 234.436} C_DIS
LIN {X 0.142,Y -457.599,Z 1292.099,A 0.000,B 0.000,C 90.000,E1 233.783} C_DIS
LIN {X -0.019,Y -457.690,Z 1292.094,A 0.000,B 0.000,C 90.000,E1 232.844} C_DIS
LIN {X -0.178,Y -457.477,Z 1292.088,A 0.000,B 0.000,C 90.000,E1 231.904} C_DIS
LIN {X -0.220,Y -456.693,Z 1292.078,A 0.000,B 0.000,C 90.000,E1 229.989} C_DIS
LIN {X 0.030,Y -456.019,Z 1292.065,A 0.000,B 0.000,C 90.000,E1 227.715} C_DIS
LIN {X -0.076,Y -455.414,Z 1292.051,A 0.000,B 0.000,C 90.000,E1 225.162} C_DIS
LIN {X 0.211,Y -455.557,Z 1292.031,A 0.000,B 0.000,C 90.000,E1 221.595} C_DIS
LIN {X 0.260,Y -456.827,Z 1292.013,A 0.000,B 0.000,C 90.000,E1 218.382} C_DIS
LIN {X -0.126,Y -458.821,Z 1291.996,A 0.000,B 0.000,C 90.000,E1 215.231} C_DIS
LIN {X 0.052,Y -461.600,Z 1291.980,A 0.000,B 0.000,C 90.000,E1 212.339} C_DIS
LIN {X -0.186,Y -463.746,Z 1291.969,A 0.000,B 0.000,C 90.000,E1 210.463} C_DIS
LIN {X 0.086,Y -466.869,Z 1291.955,A 0.000,B 0.000,C 90.000,E1 207.897} C_DIS
LIN {X -0.141,Y -469.848,Z 1291.943,A 0.000,B 0.000,C 90.000,E1 205.720} C_DIS
LIN {X 0.017,Y -472.174,Z 1291.934,A 0.000,B 0.000,C 90.000,E1 204.131} C_DIS
LIN {X -0.070,Y -475.826,Z 1291.920,A 0.000,B 0.000,C 90.000,E1 201.642} C_DIS
LIN {X 0.067,Y -479.266,Z 1291.908,A 0.000,B 0.000,C 90.000,E1 199.450} C_DIS
LIN {X 0.145,Y -482.790,Z 1291.896,A 0.000,B 0.000,C 90.000,E1 197.275} C_DIS
LIN {X 0.172,Y -485.379,Z 1291.888,A 0.000,B 0.000,C 90.000,E1 195.733} C_DIS
LIN {X 0.255,Y -488.455,Z 1291.877,A 0.000,B 0.000,C 90.000,E1 193.883} C_DIS
LIN {X -0.208,Y -491.045,Z 1291.869,A 0.000,B 0.000,C 90.000,E1 192.411} C_DIS
LIN {X 0.040,Y -494.589,Z 1291.857,A 0.000,B 0.000,C 90.000,E1 190.254} C_DIS
LIN {X -0.099,Y -497.708,Z 1291.847,A 0.000,B 0.000,C 90.000,E1 188.454} C_DIS
LIN {X -0.015,Y -499.693,Z 1291.840,A 0.000,B 0.000,C 90.000,E1 187.239} C_DIS
LIN {X -0.122,Y -502.685,Z 1291.830,A 0.000,B 0.000,C 90.000,E1 185.448} C_DIS
LIN {X 0.133,Y -505.956,Z 1291.819,A 0.000,B 0.000,C 90.000,E1 183.326} C_DIS
LIN {X 0.152,Y -508.143,Z 1291.810,A 0.000,B 0.000,C 90.000,E1 181.835} C_DIS
LIN {X -0.121,Y -509.368,Z 1291.805,A 0.000,B 0.000,C 90.000,E1 180.974} C_DIS
LIN {X -0.057,Y -511.246,Z 1291.797,A 0.000,B 0.000,C 90.000,E1 179.484} C_DIS
LIN {X 0.118,Y -512.572,Z 1291.791,A 0.000,B 0.000,C 90.000,E1 178.282} C_DIS
LIN {X -0.187,Y -513.827,Z 1291.784,A 0.000,B 0.000,C 90.000,E1 177.135} C_DIS
LIN {X 0.074,Y -514.821,Z 1291.777,A 0.000,B 0.000,C 90.000,E1 175.927} C_DIS
LIN {X -0.199,Y -515.571,Z 1291.771,A 0.000,B 0.000,C 90.000,E1 174.780} C_DIS
LIN {X 0.091,Y -516.037,Z 1291.764,A 0.000,B 0.000,C 90.000,E1 173.571} C_DIS
LIN {X -0.043,Y -516.246,Z 1291.760,A 0.000,B 0.000,C 90.000,E1 172.704} C_DIS
LIN {X -0.173,Y -516.291,Z 1291.755,A 0.000,B 0.000,C 90.000,E1 171.837} C_DIS
LIN {X 0.204,Y -516.168,Z 1291.750,A 0.000,B 0.000,C 90.000,E1 170.914} C_DIS
LIN {X 0.135,Y -515.686,Z 1291.743,A 0.000,B 0.000,C 90.000,E1 169.746} C_DIS
LIN {X 0.084,Y -515.132,Z 1291.738,A 0.000,B 0.000,C 90.000,E1 168.870} C_DIS
LIN {X 0.008,Y -513.980,Z 1291.732,A 0.000,B 0.000,C 90.000,E1 167.701} C_DIS
LIN {X -0.065,Y -512.896,Z 1291.727,A 0.000,B 0.000,C 90.000,E1 166.825} C_DIS
LIN {X -0.032,Y -511.636,Z 1291.722,A 0.000,B 0.000,C 90.000,E1 165.936} C_DIS
LIN {X -0.052,Y -509.732,Z 1291.715,A 0.000,B 0.000,C 90.000,E1 164.755} C_DIS
LIN {X -0.021,Y -506.985,Z 1291.707,A 0.000,B 0.000,C 90.000,E1 163.268} C_DIS
LIN {X 0.103,Y -504.042,Z 1291.699,A 0.000,B 0.000,C 90.000,E1 161.764} C_DIS
LIN {X 0.182,Y -502.299,Z 1291.694,A 0.000,B 0.000,C 90.000,E1 160.859} C_DIS
LIN {X -0.137,Y -501.317,Z 1291.691,A 0.000,B 0.000,C 90.000,E1 160.296} C_DIS
LIN {X -0.017,Y -499.346,Z 1291.684,A 0.000,B 0.000,C 90.000,E1 159.082} C_DIS
LIN {X 0.185,Y -498.152,Z 1291.679,A 0.000,B 0.000,C 90.000,E1 158.156} C_DIS
LIN {X -0.149,Y -497.708,Z 1291.675,A 0.000,B 0.000,C 90.000,E1 157.592} C_DIS
LIN {X -0.025,Y -497.576,Z 1291.672,A 0.000,B 0.000,C 90.000,E1 156.975} C_DIS
LIN {X 0.095,Y -497.876,Z 1291.669,A 0.000,B 0.000,C 90.000,E1 156.357} C_DIS
LIN {X 0.154,Y -498.475,Z 1291.667,A 0.000,B 0.000,C 90.000,E1 156.049} C_DIS
LIN {X -0.242,Y -499.251,Z 1291.665,A 0.000,B 0.000,C 90.000,E1 155.793} C_DIS
LIN {X -0.182,Y -500.205,Z 1291.664,A 0.000,B 0.000,C 90.000,E1 155.485} C_DIS
LIN {X -0.103,Y -502.019,Z 1291.661,A 0.000,B 0.000,C 90.000,E1 155.025} C_DIS
LIN {X -0.033,Y -503.610,Z 1291.660,A 0.000,B 0.000,C 90.000,E1 154.717} C_DIS
LIN {X -0.053,Y -506.079,Z 1291.658,A 0.000,B 0.000,C 90.000,E1 154.409} C_DIS
LIN {X 0.029,Y -508.025,Z 1291.656,A 0.000,B 0.000,C 90.000,E1 154.101} C_DIS
LIN {X 0.156,Y -509.625,Z 1291.655,A 0.000,B 0.000,C 90.000,E1 153.896} C_DIS
LIN {X 0.226,Y -514.458,Z 1291.652,A 0.000,B 0.000,C 90.000,E1 153.384} C_DIS
LIN {X -0.018,Y -523.880,Z 1291.645,A 0.000,B 0.000,C 90.000,E1 152.103} C_DIS
LIN {X 0.214,Y -527.178,Z 1291.643,A 0.000,B 0.000,C 90.000,E1 151.641} C_DIS
LIN {X -0.251,Y -530.611,Z 1291.640,A 0.000,B 0.000,C 90.000,E1 151.257} C_DIS
LIN {X 0.021,Y -533.775,Z 1291.638,A 0.000,B 0.000,C 90.000,E1 150.795} C_DIS
LIN {X 0.127,Y -535.715,Z 1291.636,A 0.000,B 0.000,C 90.000,E1 150.539} C_DIS
LIN {X 0.103,Y -537.687,Z 1291.635,A 0.000,B 0.000,C 90.000,E1 150.255} C_DIS
LIN {X 0.031,Y -545.218,Z 1291.631,A 0.000,B 0.000,C 90.000,E1 149.587} C_DIS
LIN {X 0.038,Y -557.253,Z 1291.626,A 0.000,B 0.000,C 90.000,E1 148.663} C_DIS
LIN {X -0.161,Y -564.410,Z 1291.623,A 0.000,B 0.000,C 90.000,E1 148.122} C_DIS
LIN {X 0.200,Y -578.453,Z 1291.616,A 0.000,B 0.000,C 90.000,E1 146.914} C_DIS
LIN {X 0.075,Y -583.967,Z 1291.614,A 0.000,B 0.000,C 90.000,E1 146.453} C_DIS
LIN {X -0.265,Y -590.472,Z 1291.610,A 0.000,B 0.000,C 90.000,E1 145.881} C_DIS
LIN {X -0.113,Y -595.410,Z 1291.608,A 0.000,B 0.000,C 90.000,E1 145.388} C_DIS
LIN {X -0.147,Y -600.106,Z 1291.605,A 0.000,B 0.000,C 90.000,E1 144.895} C_DIS
LIN {X -0.143,Y -605.404,Z 1291.602,A 0.000,B 0.000,C 90.000,E1 144.276} C_DIS
LIN {X -0.171,Y -608.407,Z 1291.599,A 0.000,B 0.000,C 90.000,E1 143.909} C_DIS
LIN {X -0.138,Y -612.054,Z 1291.597,A 0.000,B 0.000,C 90.000,E1 143.417} C_DIS
LIN {X -0.172,Y -615.459,Z 1291.594,A 0.000,B 0.000,C 90.000,E1 142.924} C_DIS
LIN {X -0.398,Y -618.082,Z 1291.592,A 0.000,B 0.000,C 90.000,E1 142.557} C_DIS
LIN {X 0.065,Y -622.889,Z 1291.588,A 0.000,B 0.000,C 90.000,E1 141.743} C_DIS
LIN {X -0.121,Y -625.141,Z 1291.585,A 0.000,B 0.000,C 90.000,E1 141.376} C_DIS
LIN {X 0.025,Y -629.313,Z 1291.581,A 0.000,B 0.000,C 90.000,E1 140.598} C_DIS
LIN {X -0.245,Y -634.227,Z 1291.576,A 0.000,B 0.000,C 90.000,E1 139.622} C_DIS
LIN {X -0.093,Y -637.751,Z 1291.571,A 0.000,B 0.000,C 90.000,E1 138.852} C_DIS
LIN {X -0.076,Y -643.054,Z 1291.564,A 0.000,B 0.000,C 90.000,E1 137.595} C_DIS
LIN {X 0.101,Y -647.047,Z 1291.559,A 0.000,B 0.000,C 90.000,E1 136.581} C_DIS
LIN {X 0.226,Y -652.863,Z 1291.551,A 0.000,B 0.000,C 90.000,E1 135.081} C_DIS
LIN {X 0.059,Y -656.703,Z 1291.545,A 0.000,B 0.000,C 90.000,E1 134.109} C_DIS
LIN {X 0.373,Y -662.407,Z 1291.537,A 0.000,B 0.000,C 90.000,E1 132.609} C_DIS
LIN {X -0.142,Y -666.998,Z 1291.530,A 0.000,B 0.000,C 90.000,E1 131.434} C_DIS
LIN {X -0.093,Y -671.370,Z 1291.523,A 0.000,B 0.000,C 90.000,E1 130.216} C_DIS
LIN {X 0.118,Y -675.406,Z 1291.517,A 0.000,B 0.000,C 90.000,E1 128.991} C_DIS
LIN {X -0.125,Y -679.174,Z 1291.510,A 0.000,B 0.000,C 90.000,E1 127.810} C_DIS
LIN {X 0.225,Y -682.701,Z 1291.503,A 0.000,B 0.000,C 90.000,E1 126.583} C_DIS
LIN {X -0.142,Y -684.000,Z 1291.501,A 0.000,B 0.000,C 90.000,E1 126.137} C_DIS
LIN {X -0.126,Y -687.068,Z 1291.494,A 0.000,B 0.000,C 90.000,E1 124.945} C_DIS
LIN {X -0.083,Y -689.268,Z 1291.489,A 0.000,B 0.000,C 90.000,E1 123.992} C_DIS
LIN {X -0.220,Y -690.786,Z 1291.485,A 0.000,B 0.000,C 90.000,E1 123.293} C_DIS
LIN {X 0.104,Y -692.970,Z 1291.478,A 0.000,B 0.000,C 90.000,E1 122.084} C_DIS
LIN {X 0.118,Y -695.210,Z 1291.470,A 0.000,B 0.000,C 90.000,E1 120.669} C_DIS
LIN {X -0.339,Y -696.316,Z 1291.467,A 0.000,B 0.000,C 90.000,E1 120.001} C_DIS
LIN {X -0.274,Y -697.900,Z 1291.460,A 0.000,B 0.000,C 90.000,E1 118.821} C_DIS
LIN {X -0.100,Y -698.636,Z 1291.456,A 0.000,B 0.000,C 90.000,E1 118.103} C_DIS
LIN {X 0.347,Y -699.350,Z 1291.451,A 0.000,B 0.000,C 90.000,E1 117.129} C_DIS
LIN {X -0.141,Y -699.539,Z 1291.446,A 0.000,B 0.000,C 90.000,E1 116.232} C_DIS
LIN {X 0.398,Y -699.471,Z 1291.443,A 0.000,B 0.000,C 90.000,E1 115.720} C_DIS
LIN {X 0.273,Y -699.040,Z 1291.439,A 0.000,B 0.000,C 90.000,E1 115.027} C_DIS
LIN {X -0.094,Y -698.855,Z 1291.438,A 0.000,B 0.000,C 90.000,E1 114.823} C_DIS
LIN {X 0.145,Y -698.052,Z 1291.435,A 0.000,B 0.000,C 90.000,E1 114.335} C_DIS
LIN {X -0.228,Y -697.476,Z 1291.434,A 0.000,B 0.000,C 90.000,E1 114.131} C_DIS
LIN {X 0.008,Y -695.760,Z 1291.431,A 0.000,B 0.000,C 90.000,E1 113.643} C_DIS
LIN {X 0.135,Y -695.153,Z 1291.431,A 0.000,B 0.000,C 90.000,E1 113.515} C_DIS
LIN {X -0.279,Y -691.889,Z 1291.428,A 0.000,B 0.000,C 90.000,E1 113.078} C_DIS
LIN {X -0.158,Y -690.864,Z 1291.427,A 0.000,B 0.000,C 90.000,E1 112.950} C_DIS
LIN {X -0.040,Y -689.306,Z 1291.427,A 0.000,B 0.000,C 90.000,E1 112.823} C_DIS
LIN {X 0.102,Y -684.398,Z 1291.425,A 0.000,B 0.000,C 90.000,E1 112.514} C_DIS
LIN {X -0.131,Y -681.635,Z 1291.424,A 0.000,B 0.000,C 90.000,E1 112.386} C_DIS
LIN {X 0.143,Y -679.031,Z 1291.424,A 0.000,B 0.000,C 90.000,E1 112.280} C_DIS
LIN {X 0.044,Y -674.895,Z 1291.423,A 0.000,B 0.000,C 90.000,E1 112.206} C_DIS
LIN {X -0.177,Y -672.050,Z 1291.423,A 0.000,B 0.000,C 90.000,E1 112.153} C_DIS
LIN {X 0.268,Y -669.735,Z 1291.423,A 0.000,B 0.000,C 90.000,E1 112.078} C_DIS
LIN {X 0.302,Y -663.196,Z 1291.423,A 0.000,B 0.000,C 90.000,E1 112.025} C_DIS
LIN {X 0.244,Y -645.620,Z 1291.422,A 0.000,B 0.000,C 90.000,E1 112.025} C_DIS
LIN {X 0.044,Y -643.234,Z 1291.422,A 0.000,B 0.000,C 90.000,E1 112.025} C_DIS
LIN {X 0.236,Y -638.836,Z 1291.422,A 0.000,B 0.000,C 90.000,E1 111.897} C_DIS
LIN {X 0.187,Y -638.833,Z 1291.422,A 0.000,B 0.000,C 90.000,E1 111.897} C_DIS
LIN {X -0.286,Y -639.816,Z 1291.421,A 0.000,B 0.000,C 90.000,E1 111.716} C_DIS
LIN {X -0.249,Y -641.655,Z 1291.419,A 0.000,B 0.000,C 90.000,E1 111.408} C_DIS
LIN {X 0.136,Y -649.163,Z 1291.413,A 0.000,B 0.000,C 90.000,E1 110.375} C_DIS
LIN {X 0.249,Y -651.639,Z 1291.411,A 0.000,B 0.000,C 90.000,E1 109.993} C_DIS
LIN {X 0.191,Y -654.802,Z 1291.408,A 0.000,B 0.000,C 90.000,E1 109.504} C_DIS
LIN {X -0.134,Y -659.414,Z 1291.404,A 0.000,B 0.000,C 90.000,E1 108.671} C_DIS
LIN {X -0.249,Y -662.877,Z 1291.400,A 0.000,B 0.000,C 90.000,E1 107.946} C_DIS
LIN {X -0.336,Y -665.882,Z 1291.396,A 0.000,B 0.000,C 90.000,E1 107.221} C_DIS
LIN {X 0.324,Y -667.731,Z 1291.393,A 0.000,B 0.000,C 90.000,E1 106.677} C_DIS
LIN {X 0.094,Y -670.073,Z 1291.389,A 0.000,B 0.000,C 90.000,E1 105.969} C_DIS
LIN {X 0.067,Y -671.942,Z 1291.385,A 0.000,B 0.000,C 90.000,E1 105.245} C_DIS
LIN {X -0.121,Y -673.549,Z 1291.381,A 0.000,B 0.000,C 90.000,E1 104.537} C_DIS
LIN {X -0.236,Y -674.395,Z 1291.378,A 0.000,B 0.000,C 90.000,E1 104.064} C_DIS
LIN {X 0.257,Y -675.378,Z 1291.374,A 0.000,B 0.000,C 90.000,E1 103.300} C_DIS
LIN {X 0.103,Y -676.001,Z 1291.370,A 0.000,B 0.000,C 90.000,E1 102.591} C_DIS
LIN {X -0.052,Y -676.168,Z 1291.366,A 0.000,B 0.000,C 90.000,E1 101.883} C_DIS
LIN {X -0.291,Y -676.069,Z 1291.363,A 0.000,B 0.000,C 90.000,E1 101.422} C_DIS
LIN {X 0.267,Y -675.807,Z 1291.361,A 0.000,B 0.000,C 90.000,E1 100.894} C_DIS
LIN {X 0.034,Y -675.360,Z 1291.358,A 0.000,B 0.000,C 90.000,E1 100.433} C_DIS
LIN {X -0.078,Y -674.682,Z 1291.355,A 0.000,B 0.000,C 90.000,E1 99.962} C_DIS
LIN {X -0.313,Y -673.719,Z 1291.353,A 0.000,B 0.000,C 90.000,E1 99.500} C_DIS
LIN {X 0.221,Y -672.454,Z 1291.350,A 0.000,B 0.000,C 90.000,E1 98.973} C_DIS
LIN {X 0.048,Y -671.768,Z 1291.349,A 0.000,B 0.000,C 90.000,E1 98.746} C_DIS
LIN {X -0.101,Y -670.048,Z 1291.346,A 0.000,B 0.000,C 90.000,E1 98.276} C_DIS
LIN {X 0.303,Y -667.986,Z 1291.343,A 0.000,B 0.000,C 90.000,E1 97.757} C_DIS
LIN {X -0.057,Y -665.022,Z 1291.340,A 0.000,B 0.000,C 90.000,E1 97.182} C_DIS
LIN {X 0.201,Y -660.840,Z 1291.336,A 0.000,B 0.000,C 90.000,E1 96.429} C_DIS
LIN {X -0.117,Y -657.718,Z 1291.333,A 0.000,B 0.000,C 90.000,E1 95.967} C_DIS
LIN {X 0.136,Y -654.253,Z 1291.330,A 0.000,B 0.000,C 90.000,E1 95.454} C_DIS
LIN {X -0.325,Y -649.479,Z 1291.327,A 0.000,B 0.000,C 90.000,E1 94.878} C_DIS
LIN {X -0.064,Y -645.311,Z 1291.324,A 0.000,B 0.000,C 90.000,E1 94.359} C_DIS
LIN {X 0.042,Y -639.507,Z 1291.321,A 0.000,B 0.000,C 90.000,E1 93.726} C_DIS
LIN {X 0.148,Y -633.389,Z 1291.317,A 0.000,B 0.000,C 90.000,E1 93.094} C_DIS
LIN {X 0.166,Y -624.681,Z 1291.313,A 0.000,B 0.000,C 90.000,E1 92.236} C_DIS
LIN {X -0.071,Y -618.055,Z 1291.309,A 0.000,B 0.000,C 90.000,E1 91.661} C_DIS
LIN {X -0.124,Y -615.214,Z 1291.308,A 0.000,B 0.000,C 90.000,E1 91.432} C_DIS
LIN {X 0.186,Y -609.196,Z 1291.306,A 0.000,B 0.000,C 90.000,E1 90.974} C_DIS
LIN {X 0.100,Y -602.825,Z 1291.303,A 0.000,B 0.000,C 90.000,E1 90.573} C_DIS
LIN {X -0.223,Y -596.294,Z 1291.301,A 0.000,B 0.000,C 90.000,E1 90.229} C_DIS
LIN {X -0.151,Y -589.357,Z 1291.299,A 0.000,B 0.000,C 90.000,E1 89.885} C_DIS
LIN {X -0.160,Y -582.154,Z 1291.298,A 0.000,B 0.000,C 90.000,E1 89.599} C_DIS
LIN {X 0.190,Y -576.492,Z 1291.297,A 0.000,B 0.000,C 90.000,E1 89.370} C_DIS
LIN {X -0.220,Y -573.114,Z 1291.296,A 0.000,B 0.000,C 90.000,E1 89.255} C_DIS
LIN {X 0.275,Y -571.935,Z 1291.295,A 0.000,B 0.000,C 90.000,E1 89.141} C_DIS
LIN {X 0.266,Y -570.035,Z 1291.294,A 0.000,B 0.000,C 90.000,E1 88.969} C_DIS
LIN {X 0.228,Y -570.017,Z 1291.294,A 0.000,B 0.000,C 90.000,E1 88.969} C_DIS
LIN {X -0.191,Y -569.539,Z 1291.293,A 0.000,B 0.000,C 90.000,E1 88.740} C_DIS
LIN {X -0.140,Y -569.713,Z 1291.289,A 0.000,B 0.000,C 90.000,E1 88.051} C_DIS
LIN {X 0.239,Y -572.295,Z 1291.272,A 0.000,B 0.000,C 90.000,E1 85.008} C_DIS
LIN {X -0.216,Y -574.705,Z 1291.260,A 0.000,B 0.000,C 90.000,E1 82.875} C_DIS
LIN {X -0.181,Y -576.996,Z 1291.250,A 0.000,B 0.000,C 90.000,E1 80.971} C_DIS
LIN {X 0.103,Y -578.264,Z 1291.244,A 0.000,B 0.000,C 90.000,E1 79.859} C_DIS
LIN {X -0.041,Y -579.627,Z 1291.236,A 0.000,B 0.000,C 90.000,E1 78.522} C_DIS
LIN {X -0.051,Y -580.856,Z 1291.229,A 0.000,B 0.000,C 90.000,E1 77.173} C_DIS
LIN {X -0.047,Y -581.977,Z 1291.221,A 0.000,B 0.000,C 90.000,E1 75.825} C_DIS
LIN {X 0.111,Y -582.972,Z 1291.214,A 0.000,B 0.000,C 90.000,E1 74.464} C_DIS
LIN {X -0.172,Y -583.532,Z 1291.209,A 0.000,B 0.000,C 90.000,E1 73.685} C_DIS
LIN {X 0.242,Y -584.748,Z 1291.199,A 0.000,B 0.000,C 90.000,E1 71.764} C_DIS
LIN {X 0.168,Y -585.288,Z 1291.194,A 0.000,B 0.000,C 90.000,E1 70.967} C_DIS
LIN {X -0.078,Y -586.500,Z 1291.182,A 0.000,B 0.000,C 90.000,E1 68.847} C_DIS
LIN {X 0.343,Y -587.803,Z 1291.171,A 0.000,B 0.000,C 90.000,E1 66.666} C_DIS
LIN {X 0.069,Y -588.790,Z 1291.163,A 0.000,B 0.000,C 90.000,E1 65.357} C_DIS
LIN {X -0.266,Y -590.392,Z 1291.151,A 0.000,B 0.000,C 90.000,E1 63.256} C_DIS
LIN {X -0.009,Y -592.285,Z 1291.140,A 0.000,B 0.000,C 90.000,E1 61.101} C_DIS
LIN {X -0.112,Y -594.162,Z 1291.129,A 0.000,B 0.000,C 90.000,E1 59.253} C_DIS
LIN {X -0.091,Y -595.759,Z 1291.120,A 0.000,B 0.000,C 90.000,E1 57.661} C_DIS
LIN {X -0.127,Y -597.163,Z 1291.113,A 0.000,B 0.000,C 90.000,E1 56.342} C_DIS
LIN {X -0.130,Y -598.522,Z 1291.106,A 0.000,B 0.000,C 90.000,E1 55.022} C_DIS
LIN {X 0.124,Y -599.983,Z 1291.097,A 0.000,B 0.000,C 90.000,E1 53.417} C_DIS
LIN {X -0.319,Y -601.547,Z 1291.087,A 0.000,B 0.000,C 90.000,E1 51.618} C_DIS
LIN {X 0.206,Y -602.349,Z 1291.081,A 0.000,B 0.000,C 90.000,E1 50.517} C_DIS
LIN {X 0.317,Y -603.198,Z 1291.072,A 0.000,B 0.000,C 90.000,E1 48.933} C_DIS
LIN {X -0.050,Y -603.591,Z 1291.066,A 0.000,B 0.000,C 90.000,E1 47.919} C_DIS
LIN {X 0.050,Y -604.053,Z 1291.057,A 0.000,B 0.000,C 90.000,E1 46.338} C_DIS
LIN {X -0.074,Y -604.156,Z 1291.050,A 0.000,B 0.000,C 90.000,E1 45.040} C_DIS
LIN {X 0.418,Y -604.077,Z 1291.044,A 0.000,B 0.000,C 90.000,E1 43.947} C_DIS
LIN {X 0.063,Y -603.805,Z 1291.039,A 0.000,B 0.000,C 90.000,E1 42.933} C_DIS
LIN {X -0.294,Y -603.529,Z 1291.033,A 0.000,B 0.000,C 90.000,E1 41.919} C_DIS
LIN {X 0.398,Y -603.213,Z 1291.028,A 0.000,B 0.000,C 90.000,E1 41.067} C_DIS
LIN {X 0.172,Y -602.225,Z 1291.017,A 0.000,B 0.000,C 90.000,E1 38.991} C_DIS
LIN {X -0.016,Y -601.670,Z 1291.012,A 0.000,B 0.000,C 90.000,E1 38.222} C_DIS
LIN {X 0.136,Y -600.738,Z 1291.007,A 0.000,B 0.000,C 90.000,E1 37.156} C_DIS
LIN {X 0.039,Y -599.211,Z 1290.999,A 0.000,B 0.000,C 90.000,E1 35.851} C_DIS
LIN {X -0.188,Y -597.689,Z 1290.993,A 0.000,B 0.000,C 90.000,E1 34.818} C_DIS
LIN {X 0.172,Y -596.294,Z 1290.989,A 0.000,B 0.000,C 90.000,E1 33.992} C_DIS
LIN {X -0.087,Y -594.233,Z 1290.983,A 0.000,B 0.000,C 90.000,E1 32.959} C_DIS
LIN {X 0.233,Y -592.324,Z 1290.979,A 0.000,B 0.000,C 90.000,E1 32.133} C_DIS
LIN {X 0.217,Y -590.146,Z 1290.974,A 0.000,B 0.000,C 90.000,E1 31.337} C_DIS
LIN {X 0.184,Y -587.682,Z 1290.970,A 0.000,B 0.000,C 90.000,E1 30.541} C_DIS
LIN {X 0.126,Y -584.789,Z 1290.965,A 0.000,B 0.000,C 90.000,E1 29.745} C_DIS
LIN {X 0.165,Y -582.643,Z 1290.962,A 0.000,B 0.000,C 90.000,E1 29.205} C_DIS
LIN {X -0.161,Y -579.597,Z 1290.959,A 0.000,B 0.000,C 90.000,E1 28.565} C_DIS
LIN {X -0.165,Y -577.021,Z 1290.956,A 0.000,B 0.000,C 90.000,E1 28.025} C_DIS
LIN {X -0.028,Y -573.474,Z 1290.952,A 0.000,B 0.000,C 90.000,E1 27.334} C_DIS
LIN {X -0.003,Y -571.148,Z 1290.950,A 0.000,B 0.000,C 90.000,E1 26.924} C_DIS
LIN {X 0.084,Y -566.986,Z 1290.946,A 0.000,B 0.000,C 90.000,E1 26.232} C_DIS
LIN {X 0.140,Y -562.583,Z 1290.942,A 0.000,B 0.000,C 90.000,E1 25.540} C_DIS
LIN {X 0.056,Y -556.760,Z 1290.937,A 0.000,B 0.000,C 90.000,E1 24.719} C_DIS
LIN {X 0.135,Y -552.587,Z 1290.934,A 0.000,B 0.000,C 90.000,E1 24.155} C_DIS
LIN {X 0.183,Y -548.083,Z 1290.931,A 0.000,B 0.000,C 90.000,E1 23.590} C_DIS
LIN {X -0.185,Y -539.639,Z 1290.926,A 0.000,B 0.000,C 90.000,E1 22.642} C_DIS
LIN {X 0.264,Y -534.593,Z 1290.923,A 0.000,B 0.000,C 90.000,E1 22.025} C_DIS
LIN {X -0.113,Y -525.629,Z 1290.917,A 0.000,B 0.000,C 90.000,E1 21.099} C_DIS
LIN {X 0.123,Y -519.002,Z 1290.913,A 0.000,B 0.000,C 90.000,E1 20.375} C_DIS
LIN {X -0.183,Y -510.789,Z 1290.909,A 0.000,B 0.000,C 90.000,E1 19.577} C_DIS
LIN {X 0.146,Y -503.923,Z 1290.905,A 0.000,B 0.000,C 90.000,E1 18.852} C_DIS
LIN {X -0.148,Y -494.193,Z 1290.900,A 0.000,B 0.000,C 90.000,E1 17.928} C_DIS
LIN {X 0.021,Y -484.375,Z 1290.894,A 0.000,B 0.000,C 90.000,E1 16.985} C_DIS
LIN {X 0.225,Y -474.002,Z 1290.889,A 0.000,B 0.000,C 90.000,E1 16.024} C_DIS
LIN {X -0.049,Y -463.726,Z 1290.884,A 0.000,B 0.000,C 90.000,E1 15.134} C_DIS
LIN {X -0.028,Y -447.664,Z 1290.876,A 0.000,B 0.000,C 90.000,E1 13.647} C_DIS
LIN {X 0.089,Y -426.026,Z 1290.864,A 0.000,B 0.000,C 90.000,E1 11.478} C_DIS
LIN {X 0.016,Y -407.526,Z 1290.853,A 0.000,B 0.000,C 90.000,E1 9.500} C_DIS
LIN {X 0.116,Y -400.406,Z 1290.848,A 0.000,B 0.000,C 90.000,E1 8.681} C_DIS
LIN {X -0.109,Y -396.318,Z 1290.845,A 0.000,B 0.000,C 90.000,E1 8.163} C_DIS
LIN {X -0.096,Y -395.276,Z 1290.844,A 0.000,B 0.000,C 90.000,E1 7.936} C_DIS
LIN {X -0.135,Y -395.256,Z 1290.844,A 0.000,B 0.000,C 90.000,E1 7.936} C_DIS
LIN {X 0.122,Y -395.279,Z 1290.844,A 0.000,B 0.000,C 90.000,E1 7.871} C_DIS
LIN {X 0.083,Y -395.310,Z 1290.844,A 0.000,B 0.000,C 90.000,E1 7.871} C_DIS
LIN {X 0.165,Y -396.334,Z 1290.843,A 0.000,B 0.000,C 90.000,E1 7.701} C_DIS
LIN {X 0.021,Y -399.245,Z 1290.842,A 0.000,B 0.000,C 90.000,E1 7.466} C_DIS
LIN {X 0.090,Y -403.409,Z 1290.840,A 0.000,B 0.000,C 90.000,E1 7.182} C_DIS
LIN {X 0.101,Y -410.406,Z 1290.838,A 0.000,B 0.000,C 90.000,E1 6.777} C_DIS
LIN {X 0.210,Y -416.495,Z 1290.836,A 0.000,B 0.000,C 90.000,E1 6.372} C_DIS
LIN {X -0.045,Y -422.887,Z 1290.833,A 0.000,B 0.000,C 90.000,E1 5.967} C_DIS
LIN {X -0.132,Y -430.614,Z 1290.830,A 0.000,B 0.000,C 90.000,E1 5.391} C_DIS
LIN {X 0.202,Y -441.485,Z 1290.825,A 0.000,B 0.000,C 90.000,E1 4.473} C_DIS
LIN {X -0.047,Y -450.489,Z 1290.821,A 0.000,B 0.000,C 90.000,E1 3.726} C_DIS
LIN {X -0.017,Y -454.977,Z 1290.818,A 0.000,B 0.000,C 90.000,E1 3.326} C_DIS
LIN {X -0.220,Y -460.762,Z 1290.816,A 0.000,B 0.000,C 90.000,E1 2.808} C_DIS
LIN {X -0.158,Y -466.426,Z 1290.812,A 0.000,B 0.000,C 90.000,E1 2.236} C_DIS
LIN {X -0.079,Y -473.224,Z 1290.808,A 0.000,B 0.000,C 90.000,E1 1.489} C_DIS
LIN {X 0.239,Y -479.601,Z 1290.804,A 0.000,B 0.000,C 90.000,E1 0.688} C_DIS
LIN {X 0.241,Y -483.281,Z 1290.802,A 0.000,B 0.000,C 90.000,E1 0.229} C_DIS
LIN {X 0.010,Y -488.974,Z 1290.797,A 0.000,B 0.000,C 90.000,E1 359.484} C_DIS
LIN {X 0.023,Y -495.089,Z 1290.792,A 0.000,B 0.000,C 90.000,E1 358.568} C_DIS
LIN {X -0.062,Y -499.784,Z 1290.788,A 0.000,B 0.000,C 90.000,E1 357.822} C_DIS
LIN {X -0.126,Y -504.185,Z 1290.784,A 0.000,B 0.000,C 90.000,E1 357.078} C_DIS
LIN {X 0.181,Y -507.537,Z 1290.780,A 0.000,B 0.000,C 90.000,E1 356.445} C_DIS
LIN {X 0.219,Y -511.408,Z 1290.776,A 0.000,B 0.000,C 90.000,E1 355.698} C_DIS
LIN {X 0.209,Y -516.510,Z 1290.771,A 0.000,B 0.000,C 90.000,E1 354.666} C_DIS
LIN {X -0.207,Y -521.046,Z 1290.765,A 0.000,B 0.000,C 90.000,E1 353.685} C_DIS
LIN {X 0.011,Y -522.913,Z 1290.762,A 0.000,B 0.000,C 90.000,E1 353.223} C_DIS
LIN {X -0.045,Y -526.258,Z 1290.758,A 0.000,B 0.000,C 90.000,E1 352.356} C_DIS
LIN {X -0.065,Y -529.300,Z 1290.753,A 0.000,B 0.000,C 90.000,E1 351.489} C_DIS
LIN {X -0.057,Y -532.144,Z 1290.748,A 0.000,B 0.000,C 90.000,E1 350.622} C_DIS
LIN {X 0.070,Y -534.714,Z 1290.743,A 0.000,B 0.000,C 90.000,E1 349.746} C_DIS
LIN {X 0.174,Y -536.303,Z 1290.740,A 0.000,B 0.000,C 90.000,E1 349.162} C_DIS
LIN {X -0.108,Y -539.126,Z 1290.734,A 0.000,B 0.000,C 90.000,E1 348.049} C_DIS
LIN {X 0.101,Y -541.019,Z 1290.729,A 0.000,B 0.000,C 90.000,E1 347.173} C_DIS
LIN {X -0.201,Y -542.707,Z 1290.724,A 0.000,B 0.000,C 90.000,E1 346.353} C_DIS
LIN {X 0.171,Y -544.187,Z 1290.719,A 0.000,B 0.000,C 90.000,E1 345.463} C_DIS
LIN {X 0.120,Y -545.727,Z 1290.713,A 0.000,B 0.000,C 90.000,E1 344.338} C_DIS
LIN {X -0.086,Y -546.373,Z 1290.710,A 0.000,B 0.000,C 90.000,E1 343.795} C_DIS
LIN {X -0.113,Y -547.357,Z 1290.704,A 0.000,B 0.000,C 90.000,E1 342.670} C_DIS
LIN {X 0.200,Y -547.905,Z 1290.697,A 0.000,B 0.000,C 90.000,E1 341.511} C_DIS
LIN {X 0.095,Y -547.978,Z 1290.693,A 0.000,B 0.000,C 90.000,E1 340.678} C_DIS
LIN {X 0.164,Y -547.723,Z 1290.688,A 0.000,B 0.000,C 90.000,E1 339.826} C_DIS
LIN {X 0.167,Y -547.411,Z 1290.685,A 0.000,B 0.000,C 90.000,E1 339.263} C_DIS
LIN {X 0.230,Y -546.583,Z 1290.680,A 0.000,B 0.000,C 90.000,E1 338.411} C_DIS
LIN {X 0.232,Y -545.891,Z 1290.677,A 0.000,B 0.000,C 90.000,E1 337.847} C_DIS
LIN {X 0.000,Y -543.218,Z 1290.668,A 0.000,B 0.000,C 90.000,E1 336.177} C_DIS
LIN {X -0.001,Y -540.352,Z 1290.661,A 0.000,B 0.000,C 90.000,E1 335.049} C_DIS
LIN {X -0.076,Y -537.956,Z 1290.657,A 0.000,B 0.000,C 90.000,E1 334.204} C_DIS
LIN {X 0.073,Y -535.315,Z 1290.652,A 0.000,B 0.000,C 90.000,E1 333.332} C_DIS
LIN {X -0.335,Y -531.572,Z 1290.646,A 0.000,B 0.000,C 90.000,E1 332.231} C_DIS
LIN {X 0.226,Y -528.421,Z 1290.641,A 0.000,B 0.000,C 90.000,E1 331.307} C_DIS
